gfCNCPoint1[9691] = {X 156.3350, Y 7.0477, Z -1.3333, A 0.000, B 0.000, C 0.000 }
gfCNCPoint1[9692] = {X 157.0515, Y 6.6557, Z -1.3333, A 0.000, B 0.000, C 0.000 }
gfCNCPoint1[9693] = {X 157.8307, Y 6.4112, Z -1.3333, A 0.000, B 0.000, C 0.000 }
gfCNCPoint1[9694] = {X 158.6427, Y 6.3237, Z -1.3333, A 0.000, B 0.000, C 0.000 }
gfCNCPoint1[9695] = {X 159.3760, Y 6.3239, Z -1.3333, A 0.000, B 0.000, C 0.000 }
gfCNCPoint1[9696] = {X 160.2928, Y 6.4383, Z -1.3333, A 0.000, B 0.000, C 0.000 }
gfCNCPoint1[9697] = {X 161.1617, Y 6.7524, Z -1.3333, A 0.000, B 0.000, C 0.000 }
gfCNCPoint1[9698] = {X 161.9398, Y 7.2504, Z -1.3333, A 0.000, B 0.000, C 0.000 }
gfCNCPoint1[9699] = {X 162.5889, Y 7.9079, Z -1.3333, A 0.000, B 0.000, C 0.000 }
gfCNCPoint1[9700] = {X 163.0768, Y 8.6925, Z -1.3333, A 0.000, B 0.000, C 0.000 }
gfCNCPoint1[9701] = {X 163.3795, Y 9.5653, Z -1.3333, A 0.000, B 0.000, C 0.000 }
gfCNCPoint1[9702] = {X 163.4821, Y 10.4835, Z -1.3333, A 0.000, B 0.000, C 0.000 }
gfCNCPoint1[9703] = {X 163.4821, Y 17.4615, Z -1.3333, A 0.000, B 0.000, C 0.000 }
gfCNCPoint1[9704] = {X 163.3795, Y 18.3798, Z -1.3333, A 0.000, B 0.000, C 0.000 }
gfCNCPoint1[9705] = {X 163.0767, Y 19.2527, Z -1.3333, A 0.000, B 0.000, C 0.000 }
gfCNCPoint1[9706] = {X 162.5887, Y 20.0373, Z -1.3333, A 0.000, B 0.000, C 0.000 }
gfCNCPoint1[9707] = {X 161.9396, Y 20.6948, Z -1.3333, A 0.000, B 0.000, C 0.000 }
gfCNCPoint1[9708] = {X 161.1613, Y 21.1929, Z -1.3333, A 0.000, B 0.000, C 0.000 }
gfCNCPoint1[9709] = {X 160.2923, Y 21.5068, Z -1.3333, A 0.000, B 0.000, C 0.000 }
gfCNCPoint1[9710] = {X 159.3755, Y 21.6212, Z -1.3333, A 0.000, B 0.000, C 0.000 }
gfCNCPoint1[9711] = {X 158.6798, Y 21.6215, Z -1.3333, A 0.000, B 0.000, C 0.000 }
gfCNCPoint1[9712] = {X 157.8558, Y 21.5356, Z -1.3333, A 0.000, B 0.000, C 0.000 }
gfCNCPoint1[9713] = {X 157.0647, Y 21.2896, Z -1.3333, A 0.000, B 0.000, C 0.000 }
gfCNCPoint1[9714] = {X 156.3373, Y 20.8931, Z -1.3333, A 0.000, B 0.000, C 0.000 }
gfCNCPoint1[9715] = {X 155.7019, Y 20.3615, Z -1.3333, A 0.000, B 0.000, C 0.000 }
gfCNCPoint1[9716] = {X 155.1831, Y 19.7156, Z -1.3333, A 0.000, B 0.000, C 0.000 }
gfCNCPoint1[9717] = {X 152.1155, Y 19.7172, Z -1.3333, A 0.000, B 0.000, C 0.000 }
gfCNCPoint1[9718] = {X 152.1138, Y 40.9370, Z -1.3333, A 0.000, B 0.000, C 0.000 }
gfCNCPoint1[9719] = {X 152.6210, Y 41.4829, Z -1.3333, A 0.000, B 0.000, C 0.000 }
gfCNCPoint1[9720] = {X 152.7111, Y 41.5906, Z -1.3333, A 0.000, B 0.000, C 0.000 }
gfCNCPoint1[9721] = {X 153.2166, Y 42.3853, Z -1.3333, A 0.000, B 0.000, C 0.000 }
gfCNCPoint1[9722] = {X 153.5326, Y 43.2727, Z -1.3333, A 0.000, B 0.000, C 0.000 }
gfCNCPoint1[9723] = {X 153.6431, Y 44.2081, Z -1.3333, A 0.000, B 0.000, C 0.000 }
gfCNCPoint1[9724] = {X 153.6429, Y 45.0400, Z -1.3333, A 0.000, B 0.000, C 0.000 }
gfCNCPoint1[9725] = {X 153.5310, Y 45.9591, Z -1.3333, A 0.000, B 0.000, C 0.000 }
gfCNCPoint1[9726] = {X 153.2186, Y 46.8306, Z -1.3333, A 0.000, B 0.000, C 0.000 }
gfCNCPoint1[9727] = {X 152.7212, Y 47.6115, Z -1.3333, A 0.000, B 0.000, C 0.000 }
gfCNCPoint1[9728] = {X 152.0634, Y 48.2631, Z -1.3333, A 0.000, B 0.000, C 0.000 }
gfCNCPoint1[9729] = {X 151.2778, Y 48.7530, Z -1.3333, A 0.000, B 0.000, C 0.000 }
gfCNCPoint1[9730] = {X 150.4032, Y 49.0570, Z -1.3333, A 0.000, B 0.000, C 0.000 }
gfCNCPoint1[9731] = {X 149.4831, Y 49.1600, Z -1.3333, A 0.000, B 0.000, C 0.000 }
gfCNCPoint1[9732] = {X 143.0396, Y 49.1600, Z -1.3333, A 0.000, B 0.000, C 0.000 }
gfCNCPoint1[9733] = {X 142.1185, Y 49.0567, Z -1.3333, A 0.000, B 0.000, C 0.000 }
gfCNCPoint1[9734] = {X 141.2432, Y 48.7521, Z -1.3333, A 0.000, B 0.000, C 0.000 }
gfCNCPoint1[9735] = {X 140.4570, Y 48.2612, Z -1.3333, A 0.000, B 0.000, C 0.000 }
gfCNCPoint1[9736] = {X 139.7990, Y 47.6084, Z -1.3333, A 0.000, B 0.000, C 0.000 }
gfCNCPoint1[9737] = {X 139.3019, Y 46.8261, Z -1.3333, A 0.000, B 0.000, C 0.000 }
gfCNCPoint1[9738] = {X 138.9903, Y 45.9532, Z -1.3333, A 0.000, B 0.000, C 0.000 }
gfCNCPoint1[9739] = {X 138.8798, Y 45.0329, Z -1.3333, A 0.000, B 0.000, C 0.000 }
gfCNCPoint1[9740] = {X 138.8800, Y 44.1516, Z -1.3333, A 0.000, B 0.000, C 0.000 }
gfCNCPoint1[9741] = {X 138.9906, Y 43.2545, Z -1.3333, A 0.000, B 0.000, C 0.000 }
gfCNCPoint1[9742] = {X 139.2922, Y 42.4026, Z -1.3333, A 0.000, B 0.000, C 0.000 }
gfCNCPoint1[9743] = {X 139.7708, Y 41.6358, Z -1.3333, A 0.000, B 0.000, C 0.000 }
gfCNCPoint1[9744] = {X 140.4036, Y 40.9906, Z -1.3333, A 0.000, B 0.000, C 0.000 }
gfCNCPoint1[9745] = {X 140.4036, Y 30.3961, Z -1.3333, A 0.000, B 0.000, C 0.000 }
gfCNCPoint1[9746] = {X 136.4036, Y 30.3961, Z -1.3333, A 0.000, B 0.000, C 0.000 }
gfCNCPoint1[9747] = {X 140.4836, Y 30.3961, Z -1.3333, A 0.000, B 0.000, C 0.000 }
gfCNCPoint1[9748] = {X 140.4836, Y 19.6366, Z -1.3333, A 0.000, B 0.000, C 0.000 }
gfCNCPoint1[9749] = {X 137.2908, Y 19.6355, Z -1.3333, A 0.000, B 0.000, C 0.000 }
gfCNCPoint1[9750] = {X 137.2218, Y 19.7475, Z -1.3333, A 0.000, B 0.000, C 0.000 }
gfCNCPoint1[9751] = {X 136.5756, Y 20.4907, Z -1.3333, A 0.000, B 0.000, C 0.000 }
gfCNCPoint1[9752] = {X 135.7702, Y 21.0573, Z -1.3333, A 0.000, B 0.000, C 0.000 }
gfCNCPoint1[9753] = {X 134.8524, Y 21.4145, Z -1.3333, A 0.000, B 0.000, C 0.000 }
gfCNCPoint1[9754] = {X 133.8758, Y 21.5414, Z -1.3333, A 0.000, B 0.000, C 0.000 }
gfCNCPoint1[9755] = {X 133.2006, Y 21.5415, Z -1.3333, A 0.000, B 0.000, C 0.000 }
gfCNCPoint1[9756] = {X 132.2928, Y 21.4392, Z -1.3333, A 0.000, B 0.000, C 0.000 }
gfCNCPoint1[9757] = {X 131.4304, Y 21.1375, Z -1.3333, A 0.000, B 0.000, C 0.000 }
gfCNCPoint1[9758] = {X 130.6568, Y 20.6514, Z -1.3333, A 0.000, B 0.000, C 0.000 }
gfCNCPoint1[9759] = {X 130.0108, Y 20.0054, Z -1.3333, A 0.000, B 0.000, C 0.000 }
gfCNCPoint1[9760] = {X 129.5247, Y 19.2318, Z -1.3333, A 0.000, B 0.000, C 0.000 }
gfCNCPoint1[9761] = {X 129.2229, Y 18.3694, Z -1.3333, A 0.000, B 0.000, C 0.000 }
gfCNCPoint1[9762] = {X 129.1206, Y 17.4615, Z -1.3333, A 0.000, B 0.000, C 0.000 }
gfCNCPoint1[9763] = {X 129.1206, Y 10.4835, Z -1.3333, A 0.000, B 0.000, C 0.000 }
gfCNCPoint1[9764] = {X 129.2215, Y 9.5820, Z -1.3333, A 0.000, B 0.000, C 0.000 }
gfCNCPoint1[9765] = {X 129.5191, Y 8.7250, Z -1.3333, A 0.000, B 0.000, C 0.000 }
gfCNCPoint1[9766] = {X 129.9986, Y 7.9550, Z -1.3333, A 0.000, B 0.000, C 0.000 }
gfCNCPoint1[9767] = {X 130.6365, Y 7.3099, Z -1.3333, A 0.000, B 0.000, C 0.000 }
gfCNCPoint1[9768] = {X 131.4011, Y 6.8218, Z -1.3333, A 0.000, B 0.000, C 0.000 }
gfCNCPoint1[9769] = {X 132.2547, Y 6.5147, Z -1.3333, A 0.000, B 0.000, C 0.000 }
gfCNCPoint1[9770] = {X 133.1551, Y 6.4038, Z -1.3333, A 0.000, B 0.000, C 0.000 }
gfCNCPoint1[9771] = {X 133.8841, Y 6.4037, Z -1.3333, A 0.000, B 0.000, C 0.000 }
gfCNCPoint1[9772] = {X 134.6877, Y 6.4920, Z -1.3333, A 0.000, B 0.000, C 0.000 }
gfCNCPoint1[9773] = {X 135.4580, Y 6.7370, Z -1.3333, A 0.000, B 0.000, C 0.000 }
gfCNCPoint1[9774] = {X 136.1649, Y 7.1291, Z -1.3333, A 0.000, B 0.000, C 0.000 }
gfCNCPoint1[9775] = {X 136.7806, Y 7.6528, Z -1.3333, A 0.000, B 0.000, C 0.000 }
gfCNCPoint1[9776] = {X 137.2810, Y 8.2877, Z -1.3333, A 0.000, B 0.000, C 0.000 }
gfCNCPoint1[9777] = {X 155.2410, Y 8.2888, Z -1.3333, A 0.000, B 0.000, C 0.000 }
gfCNCPoint1[9778] = {X 155.2864, Y 8.2192, Z -1.3333, A 0.000, B 0.000, C 0.000 }
gfCNCPoint1[9779] = {X 155.3332, Y 8.1507, Z -1.3333, A 0.000, B 0.000, C 0.000 }
gfCNCPoint1[9780] = {X 155.9783, Y 7.4266, Z -1.3333, A 0.000, B 0.000, C 0.000 }
gfCNCPoint1[9781] = {X 156.7761, Y 6.8752, Z -1.3333, A 0.000, B 0.000, C 0.000 }
gfCNCPoint1[9782] = {X 157.6815, Y 6.5277, Z -1.3333, A 0.000, B 0.000, C 0.000 }
gfCNCPoint1[9783] = {X 158.6434, Y 6.4037, Z -1.3333, A 0.000, B 0.000, C 0.000 }
gfCNCPoint1[9784] = {X 159.3750, Y 6.4039, Z -1.3333, A 0.000, B 0.000, C 0.000 }
gfCNCPoint1[9785] = {X 160.2741, Y 6.5161, Z -1.3333, A 0.000, B 0.000, C 0.000 }
gfCNCPoint1[9786] = {X 161.1263, Y 6.8241, Z -1.3333, A 0.000, B 0.000, C 0.000 }
gfCNCPoint1[9787] = {X 161.8895, Y 7.3126, Z -1.3333, A 0.000, B 0.000, C 0.000 }
gfCNCPoint1[9788] = {X 162.5260, Y 7.9574, Z -1.3333, A 0.000, B 0.000, C 0.000 }
gfCNCPoint1[9789] = {X 163.0046, Y 8.7269, Z -1.3333, A 0.000, B 0.000, C 0.000 }
gfCNCPoint1[9790] = {X 163.3015, Y 9.5830, Z -1.3333, A 0.000, B 0.000, C 0.000 }
gfCNCPoint1[9791] = {X 163.4021, Y 10.4835, Z -1.3333, A 0.000, B 0.000, C 0.000 }
gfCNCPoint1[9792] = {X 163.4021, Y 17.4615, Z -1.3333, A 0.000, B 0.000, C 0.000 }
gfCNCPoint1[9793] = {X 163.3015, Y 18.3621, Z -1.3333, A 0.000, B 0.000, C 0.000 }
gfCNCPoint1[9794] = {X 163.0046, Y 19.2182, Z -1.3333, A 0.000, B 0.000, C 0.000 }
gfCNCPoint1[9795] = {X 162.5260, Y 19.9876, Z -1.3333, A 0.000, B 0.000, C 0.000 }
gfCNCPoint1[9796] = {X 161.8895, Y 20.6325, Z -1.3333, A 0.000, B 0.000, C 0.000 }
gfCNCPoint1[9797] = {X 161.1263, Y 21.1209, Z -1.3333, A 0.000, B 0.000, C 0.000 }
gfCNCPoint1[9798] = {X 160.2741, Y 21.4289, Z -1.3333, A 0.000, B 0.000, C 0.000 }
gfCNCPoint1[9799] = {X 159.3750, Y 21.5412, Z -1.3333, A 0.000, B 0.000, C 0.000 }
gfCNCPoint1[9800] = {X 158.6802, Y 21.5415, Z -1.3333, A 0.000, B 0.000, C 0.000 }
gfCNCPoint1[9801] = {X 157.8634, Y 21.4555, Z -1.3333, A 0.000, B 0.000, C 0.000 }
gfCNCPoint1[9802] = {X 157.0800, Y 21.2091, Z -1.3333, A 0.000, B 0.000, C 0.000 }
gfCNCPoint1[9803] = {X 156.3609, Y 20.8123, Z -1.3333, A 0.000, B 0.000, C 0.000 }
gfCNCPoint1[9804] = {X 155.7349, Y 20.2807, Z -1.3333, A 0.000, B 0.000, C 0.000 }
gfCNCPoint1[9805] = {X 155.2267, Y 19.6356, Z -1.3333, A 0.000, B 0.000, C 0.000 }
gfCNCPoint1[9806] = {X 152.0355, Y 19.6373, Z -1.3333, A 0.000, B 0.000, C 0.000 }
gfCNCPoint1[9807] = {X 152.0338, Y 40.9684, Z -1.3333, A 0.000, B 0.000, C 0.000 }
gfCNCPoint1[9808] = {X 152.5609, Y 41.5359, Z -1.3333, A 0.000, B 0.000, C 0.000 }
gfCNCPoint1[9809] = {X 152.6492, Y 41.6414, Z -1.3333, A 0.000, B 0.000, C 0.000 }
gfCNCPoint1[9810] = {X 153.1450, Y 42.4209, Z -1.3333, A 0.000, B 0.000, C 0.000 }
gfCNCPoint1[9811] = {X 153.4548, Y 43.2911, Z -1.3333, A 0.000, B 0.000, C 0.000 }
gfCNCPoint1[9812] = {X 153.5631, Y 44.2085, Z -1.3333, A 0.000, B 0.000, C 0.000 }
gfCNCPoint1[9813] = {X 153.5629, Y 45.0392, Z -1.3333, A 0.000, B 0.000, C 0.000 }
gfCNCPoint1[9814] = {X 153.4532, Y 45.9406, Z -1.3333, A 0.000, B 0.000, C 0.000 }
gfCNCPoint1[9815] = {X 153.1468, Y 46.7954, Z -1.3333, A 0.000, B 0.000, C 0.000 }
gfCNCPoint1[9816] = {X 152.6589, Y 47.5613, Z -1.3333, A 0.000, B 0.000, C 0.000 }
gfCNCPoint1[9817] = {X 152.0138, Y 48.2003, Z -1.3333, A 0.000, B 0.000, C 0.000 }
gfCNCPoint1[9818] = {X 151.2432, Y 48.6808, Z -1.3333, A 0.000, B 0.000, C 0.000 }
gfCNCPoint1[9819] = {X 150.3855, Y 48.9789, Z -1.3333, A 0.000, B 0.000, C 0.000 }
gfCNCPoint1[9820] = {X 149.4831, Y 49.0800, Z -1.3333, A 0.000, B 0.000, C 0.000 }
gfCNCPoint1[9821] = {X 143.0396, Y 49.0800, Z -1.3333, A 0.000, B 0.000, C 0.000 }
gfCNCPoint1[9822] = {X 142.1362, Y 48.9787, Z -1.3333, A 0.000, B 0.000, C 0.000 }
gfCNCPoint1[9823] = {X 141.2777, Y 48.6799, Z -1.3333, A 0.000, B 0.000, C 0.000 }
gfCNCPoint1[9824] = {X 140.5066, Y 48.1985, Z -1.3333, A 0.000, B 0.000, C 0.000 }
gfCNCPoint1[9825] = {X 139.8613, Y 47.5582, Z -1.3333, A 0.000, B 0.000, C 0.000 }
gfCNCPoint1[9826] = {X 139.3737, Y 46.7910, Z -1.3333, A 0.000, B 0.000, C 0.000 }
gfCNCPoint1[9827] = {X 139.0682, Y 45.9349, Z -1.3333, A 0.000, B 0.000, C 0.000 }
gfCNCPoint1[9828] = {X 138.9598, Y 45.0323, Z -1.3333, A 0.000, B 0.000, C 0.000 }
gfCNCPoint1[9829] = {X 138.9600, Y 44.1527, Z -1.3333, A 0.000, B 0.000, C 0.000 }
gfCNCPoint1[9830] = {X 139.0706, Y 43.2637, Z -1.3333, A 0.000, B 0.000, C 0.000 }
gfCNCPoint1[9831] = {X 139.3725, Y 42.4203, Z -1.3333, A 0.000, B 0.000, C 0.000 }
gfCNCPoint1[9832] = {X 139.8512, Y 41.6631, Z -1.3333, A 0.000, B 0.000, C 0.000 }
gfCNCPoint1[9833] = {X 140.4836, Y 41.0287, Z -1.3333, A 0.000, B 0.000, C 0.000 }
gfCNCPoint1[9834] = {X 140.4836, Y 30.3961, Z -1.3333, A 0.000, B 0.000, C 0.000 }
gfCNCPoint1[9835] = {X 136.4836, Y 30.3961, Z -1.3333, A 0.000, B 0.000, C 0.000 }
gfCNCPoint1[9836] = {X 140.5636, Y 30.3961, Z -1.3333, A 0.000, B 0.000, C 0.000 }
gfCNCPoint1[9837] = {X 140.5636, Y 19.9565, Z -1.3333, A 0.000, B 0.000, C 0.000 }
gfCNCPoint1[9838] = {X 140.5652, Y 19.5566, Z -1.3333, A 0.000, B 0.000, C 0.000 }
gfCNCPoint1[9839] = {X 137.2663, Y 19.5555, Z -1.3333, A 0.000, B 0.000, C 0.000 }
gfCNCPoint1[9840] = {X 137.2435, Y 19.5597, Z -1.3333, A 0.000, B 0.000, C 0.000 }
gfCNCPoint1[9841] = {X 137.1376, Y 19.7289, Z -1.3333, A 0.000, B 0.000, C 0.000 }
gfCNCPoint1[9842] = {X 136.4981, Y 20.4526, Z -1.3333, A 0.000, B 0.000, C 0.000 }
gfCNCPoint1[9843] = {X 135.7038, Y 21.0020, Z -1.3333, A 0.000, B 0.000, C 0.000 }
gfCNCPoint1[9844] = {X 134.8009, Y 21.3450, Z -1.3333, A 0.000, B 0.000, C 0.000 }
gfCNCPoint1[9845] = {X 133.8421, Y 21.4615, Z -1.3333, A 0.000, B 0.000, C 0.000 }
gfCNCPoint1[9846] = {X 133.2006, Y 21.4615, Z -1.3333, A 0.000, B 0.000, C 0.000 }
gfCNCPoint1[9847] = {X 132.3106, Y 21.3612, Z -1.3333, A 0.000, B 0.000, C 0.000 }
gfCNCPoint1[9848] = {X 131.4651, Y 21.0654, Z -1.3333, A 0.000, B 0.000, C 0.000 }
gfCNCPoint1[9849] = {X 130.7067, Y 20.5889, Z -1.3333, A 0.000, B 0.000, C 0.000 }
gfCNCPoint1[9850] = {X 130.0733, Y 19.9555, Z -1.3333, A 0.000, B 0.000, C 0.000 }
gfCNCPoint1[9851] = {X 129.5968, Y 19.1971, Z -1.3333, A 0.000, B 0.000, C 0.000 }
gfCNCPoint1[9852] = {X 129.3009, Y 18.3516, Z -1.3333, A 0.000, B 0.000, C 0.000 }
gfCNCPoint1[9853] = {X 129.2006, Y 17.4615, Z -1.3333, A 0.000, B 0.000, C 0.000 }
gfCNCPoint1[9854] = {X 129.2006, Y 10.4835, Z -1.3333, A 0.000, B 0.000, C 0.000 }
gfCNCPoint1[9855] = {X 129.3009, Y 9.5934, Z -1.3333, A 0.000, B 0.000, C 0.000 }
gfCNCPoint1[9856] = {X 129.5968, Y 8.7480, Z -1.3333, A 0.000, B 0.000, C 0.000 }
gfCNCPoint1[9857] = {X 130.0733, Y 7.9895, Z -1.3333, A 0.000, B 0.000, C 0.000 }
gfCNCPoint1[9858] = {X 130.7067, Y 7.3562, Z -1.3333, A 0.000, B 0.000, C 0.000 }
gfCNCPoint1[9859] = {X 131.4651, Y 6.8796, Z -1.3333, A 0.000, B 0.000, C 0.000 }
gfCNCPoint1[9860] = {X 132.3106, Y 6.5838, Z -1.3333, A 0.000, B 0.000, C 0.000 }
gfCNCPoint1[9861] = {X 133.2007, Y 6.4835, Z -1.3333, A 0.000, B 0.000, C 0.000 }
gfCNCPoint1[9862] = {X 133.8833, Y 6.4837, Z -1.3333, A 0.000, B 0.000, C 0.000 }
gfCNCPoint1[9863] = {X 134.6796, Y 6.5721, Z -1.3333, A 0.000, B 0.000, C 0.000 }
gfCNCPoint1[9864] = {X 135.4423, Y 6.8175, Z -1.3333, A 0.000, B 0.000, C 0.000 }
gfCNCPoint1[9865] = {X 136.1408, Y 7.2099, Z -1.3333, A 0.000, B 0.000, C 0.000 }
gfCNCPoint1[9866] = {X 136.7471, Y 7.7336, Z -1.3333, A 0.000, B 0.000, C 0.000 }
gfCNCPoint1[9867] = {X 137.2369, Y 8.3677, Z -1.3333, A 0.000, B 0.000, C 0.000 }
gfCNCPoint1[9868] = {X 155.2276, Y 8.3677, Z -1.3333, A 0.000, B 0.000, C 0.000 }
gfCNCPoint1[9869] = {X 155.2814, Y 8.3748, Z -1.3333, A 0.000, B 0.000, C 0.000 }
gfCNCPoint1[9870] = {X 155.3389, Y 8.2848, Z -1.3333, A 0.000, B 0.000, C 0.000 }
gfCNCPoint1[9871] = {X 155.3988, Y 8.1964, Z -1.3333, A 0.000, B 0.000, C 0.000 }
gfCNCPoint1[9872] = {X 156.0381, Y 7.4805, Z -1.3333, A 0.000, B 0.000, C 0.000 }
gfCNCPoint1[9873] = {X 156.8296, Y 6.9374, Z -1.3333, A 0.000, B 0.000, C 0.000 }
gfCNCPoint1[9874] = {X 157.7277, Y 6.5986, Z -1.3333, A 0.000, B 0.000, C 0.000 }
gfCNCPoint1[9875] = {X 158.6806, Y 6.4835, Z -1.3333, A 0.000, B 0.000, C 0.000 }
gfCNCPoint1[9876] = {X 159.3739, Y 6.4839, Z -1.3333, A 0.000, B 0.000, C 0.000 }
gfCNCPoint1[9877] = {X 160.2554, Y 6.5939, Z -1.3333, A 0.000, B 0.000, C 0.000 }
gfCNCPoint1[9878] = {X 161.0909, Y 6.8959, Z -1.3333, A 0.000, B 0.000, C 0.000 }
gfCNCPoint1[9879] = {X 161.8391, Y 7.3747, Z -1.3333, A 0.000, B 0.000, C 0.000 }
gfCNCPoint1[9880] = {X 162.4632, Y 8.0070, Z -1.3333, A 0.000, B 0.000, C 0.000 }
gfCNCPoint1[9881] = {X 162.9324, Y 8.7613, Z -1.3333, A 0.000, B 0.000, C 0.000 }
gfCNCPoint1[9882] = {X 163.2234, Y 9.6007, Z -1.3333, A 0.000, B 0.000, C 0.000 }
gfCNCPoint1[9883] = {X 163.3221, Y 10.4835, Z -1.3333, A 0.000, B 0.000, C 0.000 }
gfCNCPoint1[9884] = {X 163.3221, Y 17.4615, Z -1.3333, A 0.000, B 0.000, C 0.000 }
gfCNCPoint1[9885] = {X 163.2218, Y 18.3516, Z -1.3333, A 0.000, B 0.000, C 0.000 }
gfCNCPoint1[9886] = {X 162.9260, Y 19.1971, Z -1.3333, A 0.000, B 0.000, C 0.000 }
gfCNCPoint1[9887] = {X 162.4494, Y 19.9555, Z -1.3333, A 0.000, B 0.000, C 0.000 }
gfCNCPoint1[9888] = {X 161.8160, Y 20.5889, Z -1.3333, A 0.000, B 0.000, C 0.000 }
gfCNCPoint1[9889] = {X 161.0576, Y 21.0654, Z -1.3333, A 0.000, B 0.000, C 0.000 }
gfCNCPoint1[9890] = {X 160.2121, Y 21.3613, Z -1.3333, A 0.000, B 0.000, C 0.000 }
gfCNCPoint1[9891] = {X 159.3221, Y 21.4615, Z -1.3333, A 0.000, B 0.000, C 0.000 }
gfCNCPoint1[9892] = {X 158.6806, Y 21.4615, Z -1.3333, A 0.000, B 0.000, C 0.000 }
gfCNCPoint1[9893] = {X 157.8711, Y 21.3754, Z -1.3333, A 0.000, B 0.000, C 0.000 }
gfCNCPoint1[9894] = {X 157.0954, Y 21.1287, Z -1.3333, A 0.000, B 0.000, C 0.000 }
gfCNCPoint1[9895] = {X 156.3848, Y 20.7315, Z -1.3333, A 0.000, B 0.000, C 0.000 }
gfCNCPoint1[9896] = {X 155.7683, Y 20.1999, Z -1.3333, A 0.000, B 0.000, C 0.000 }
gfCNCPoint1[9897] = {X 155.2709, Y 19.5555, Z -1.3333, A 0.000, B 0.000, C 0.000 }
gfCNCPoint1[9898] = {X 151.9555, Y 19.5573, Z -1.3333, A 0.000, B 0.000, C 0.000 }
gfCNCPoint1[9899] = {X 151.9538, Y 40.9999, Z -1.3333, A 0.000, B 0.000, C 0.000 }
gfCNCPoint1[9900] = {X 152.5009, Y 41.5888, Z -1.3333, A 0.000, B 0.000, C 0.000 }
gfCNCPoint1[9901] = {X 152.5874, Y 41.6922, Z -1.3333, A 0.000, B 0.000, C 0.000 }
gfCNCPoint1[9902] = {X 153.0733, Y 42.4564, Z -1.3333, A 0.000, B 0.000, C 0.000 }
gfCNCPoint1[9903] = {X 153.3769, Y 43.3096, Z -1.3333, A 0.000, B 0.000, C 0.000 }
gfCNCPoint1[9904] = {X 153.4831, Y 44.2089, Z -1.3333, A 0.000, B 0.000, C 0.000 }
gfCNCPoint1[9905] = {X 153.4829, Y 45.0384, Z -1.3333, A 0.000, B 0.000, C 0.000 }
gfCNCPoint1[9906] = {X 153.3753, Y 45.9222, Z -1.3333, A 0.000, B 0.000, C 0.000 }
gfCNCPoint1[9907] = {X 153.0750, Y 46.7602, Z -1.3333, A 0.000, B 0.000, C 0.000 }
gfCNCPoint1[9908] = {X 152.5967, Y 47.5111, Z -1.3333, A 0.000, B 0.000, C 0.000 }
gfCNCPoint1[9909] = {X 151.9642, Y 48.1376, Z -1.3333, A 0.000, B 0.000, C 0.000 }
gfCNCPoint1[9910] = {X 151.2087, Y 48.6086, Z -1.3333, A 0.000, B 0.000, C 0.000 }
gfCNCPoint1[9911] = {X 150.3678, Y 48.9009, Z -1.3333, A 0.000, B 0.000, C 0.000 }
gfCNCPoint1[9912] = {X 149.4831, Y 49.0000, Z -1.3333, A 0.000, B 0.000, C 0.000 }
gfCNCPoint1[9913] = {X 143.0396, Y 49.0000, Z -1.3333, A 0.000, B 0.000, C 0.000 }
gfCNCPoint1[9914] = {X 142.1495, Y 48.8997, Z -1.3333, A 0.000, B 0.000, C 0.000 }
gfCNCPoint1[9915] = {X 141.3041, Y 48.6039, Z -1.3333, A 0.000, B 0.000, C 0.000 }
gfCNCPoint1[9916] = {X 140.5457, Y 48.1273, Z -1.3333, A 0.000, B 0.000, C 0.000 }
gfCNCPoint1[9917] = {X 139.9123, Y 47.4939, Z -1.3333, A 0.000, B 0.000, C 0.000 }
gfCNCPoint1[9918] = {X 139.4357, Y 46.7355, Z -1.3333, A 0.000, B 0.000, C 0.000 }
gfCNCPoint1[9919] = {X 139.1399, Y 45.8900, Z -1.3333, A 0.000, B 0.000, C 0.000 }
gfCNCPoint1[9920] = {X 139.0396, Y 44.9999, Z -1.3333, A 0.000, B 0.000, C 0.000 }
gfCNCPoint1[9921] = {X 139.0400, Y 44.1538, Z -1.3333, A 0.000, B 0.000, C 0.000 }
gfCNCPoint1[9922] = {X 139.1506, Y 43.2730, Z -1.3333, A 0.000, B 0.000, C 0.000 }
gfCNCPoint1[9923] = {X 139.4528, Y 42.4382, Z -1.3333, A 0.000, B 0.000, C 0.000 }
gfCNCPoint1[9924] = {X 139.9317, Y 41.6907, Z -1.3333, A 0.000, B 0.000, C 0.000 }
gfCNCPoint1[9925] = {X 140.5636, Y 41.0672, Z -1.3333, A 0.000, B 0.000, C 0.000 }
gfCNCPoint1[9926] = {X 140.5636, Y 30.3961, Z -1.3333, A 0.000, B 0.000, C 0.000 }
gfCNCPoint1[9927] = {X 136.4836, Y 30.3961, Z -1.3333, A 0.000, B 0.000, C 0.000 }
gfCNCPoint1[9928] = {X 136.4836, Y 30.3961, Z 1.6667, A 0.000, B 0.000, C 0.000 }
gfCNCPoint1[9929] = {X 136.4836, Y 30.3961, Z 11.0000, A 0.000, B 0.000, C 0.000 }
gfCNCPoint1[9930] = {X 137.6639, Y 74.8937, Z 11.0000, A 0.000, B 0.000, C 0.000 }
gfCNCPoint1[9931] = {X 137.6639, Y 74.8937, Z 1.6667, A 0.000, B 0.000, C 0.000 }
gfCNCPoint1[9932] = {X 137.6639, Y 74.8937, Z -1.3333, A 0.000, B 0.000, C 0.000 }
gfCNCPoint1[9933] = {X 140.6806, Y 77.6408, Z -1.3333, A 0.000, B 0.000, C 0.000 }
gfCNCPoint1[9934] = {X 155.6330, Y 61.2211, Z -1.3333, A 0.000, B 0.000, C 0.000 }
gfCNCPoint1[9935] = {X 155.2777, Y 60.5151, Z -1.3333, A 0.000, B 0.000, C 0.000 }
gfCNCPoint1[9936] = {X 155.0569, Y 59.7562, Z -1.3333, A 0.000, B 0.000, C 0.000 }
gfCNCPoint1[9937] = {X 154.9781, Y 58.9697, Z -1.3333, A 0.000, B 0.000, C 0.000 }
gfCNCPoint1[9938] = {X 154.9780, Y 58.0000, Z -1.3333, A 0.000, B 0.000, C 0.000 }
gfCNCPoint1[9939] = {X 155.0863, Y 57.0387, Z -1.3333, A 0.000, B 0.000, C 0.000 }
gfCNCPoint1[9940] = {X 155.4058, Y 56.1256, Z -1.3333, A 0.000, B 0.000, C 0.000 }
gfCNCPoint1[9941] = {X 155.9204, Y 55.3065, Z -1.3333, A 0.000, B 0.000, C 0.000 }
gfCNCPoint1[9942] = {X 156.6045, Y 54.6225, Z -1.3333, A 0.000, B 0.000, C 0.000 }
gfCNCPoint1[9943] = {X 157.4236, Y 54.1078, Z -1.3333, A 0.000, B 0.000, C 0.000 }
gfCNCPoint1[9944] = {X 158.3367, Y 53.7883, Z -1.3333, A 0.000, B 0.000, C 0.000 }
gfCNCPoint1[9945] = {X 159.2980, Y 53.6800, Z -1.3333, A 0.000, B 0.000, C 0.000 }
gfCNCPoint1[9946] = {X 178.5335, Y 53.6800, Z -1.3333, A 0.000, B 0.000, C 0.000 }
gfCNCPoint1[9947] = {X 179.4948, Y 53.7883, Z -1.3333, A 0.000, B 0.000, C 0.000 }
gfCNCPoint1[9948] = {X 180.4079, Y 54.1078, Z -1.3333, A 0.000, B 0.000, C 0.000 }
gfCNCPoint1[9949] = {X 181.2270, Y 54.6225, Z -1.3333, A 0.000, B 0.000, C 0.000 }
gfCNCPoint1[9950] = {X 181.9110, Y 55.3065, Z -1.3333, A 0.000, B 0.000, C 0.000 }
gfCNCPoint1[9951] = {X 182.4257, Y 56.1256, Z -1.3333, A 0.000, B 0.000, C 0.000 }
gfCNCPoint1[9952] = {X 182.7452, Y 57.0387, Z -1.3333, A 0.000, B 0.000, C 0.000 }
gfCNCPoint1[9953] = {X 182.8535, Y 58.0000, Z -1.3333, A 0.000, B 0.000, C 0.000 }
gfCNCPoint1[9954] = {X 182.8535, Y 58.9342, Z -1.3333, A 0.000, B 0.000, C 0.000 }
gfCNCPoint1[9955] = {X 182.7807, Y 59.7236, Z -1.3333, A 0.000, B 0.000, C 0.000 }
gfCNCPoint1[9956] = {X 182.5649, Y 60.4865, Z -1.3333, A 0.000, B 0.000, C 0.000 }
gfCNCPoint1[9957] = {X 182.2134, Y 61.1970, Z -1.3333, A 0.000, B 0.000, C 0.000 }
gfCNCPoint1[9958] = {X 209.4771, Y 90.9538, Z -1.3333, A 0.000, B 0.000, C 0.000 }
gfCNCPoint1[9959] = {X 210.1356, Y 91.6218, Z -1.3333, A 0.000, B 0.000, C 0.000 }
gfCNCPoint1[9960] = {X 210.8409, Y 92.2402, Z -1.3333, A 0.000, B 0.000, C 0.000 }
gfCNCPoint1[9961] = {X 211.1176, Y 92.4147, Z -1.3333, A 0.000, B 0.000, C 0.000 }
gfCNCPoint1[9962] = {X 211.4280, Y 92.5180, Z -1.3333, A 0.000, B 0.000, C 0.000 }
gfCNCPoint1[9963] = {X 212.4217, Y 92.7023, Z -1.3333, A 0.000, B 0.000, C 0.000 }
gfCNCPoint1[9964] = {X 213.4259, Y 92.8161, Z -1.3333, A 0.000, B 0.000, C 0.000 }
gfCNCPoint1[9965] = {X 214.4655, Y 92.7370, Z -1.3333, A 0.000, B 0.000, C 0.000 }
gfCNCPoint1[9966] = {X 215.5064, Y 92.6769, Z -1.3333, A 0.000, B 0.000, C 0.000 }
gfCNCPoint1[9967] = {X 216.1767, Y 92.6037, Z -1.3333, A 0.000, B 0.000, C 0.000 }
gfCNCPoint1[9968] = {X 216.8222, Y 92.4086, Z -1.3333, A 0.000, B 0.000, C 0.000 }
gfCNCPoint1[9969] = {X 217.4210, Y 92.0984, Z -1.3333, A 0.000, B 0.000, C 0.000 }
gfCNCPoint1[9970] = {X 222.9613, Y 88.5229, Z -1.3333, A 0.000, B 0.000, C 0.000 }
gfCNCPoint1[9971] = {X 245.8295, Y 73.8994, Z -1.3333, A 0.000, B 0.000, C 0.000 }
gfCNCPoint1[9972] = {X 221.6305, Y 64.4024, Z -1.3333, A 0.000, B 0.000, C 0.000 }
gfCNCPoint1[9973] = {X 219.8632, Y 63.8108, Z -1.3333, A 0.000, B 0.000, C 0.000 }
gfCNCPoint1[9974] = {X 218.0398, Y 63.4255, Z -1.3333, A 0.000, B 0.000, C 0.000 }
gfCNCPoint1[9975] = {X 216.1843, Y 63.2516, Z -1.3333, A 0.000, B 0.000, C 0.000 }
gfCNCPoint1[9976] = {X 215.2524, Y 63.1173, Z -1.3333, A 0.000, B 0.000, C 0.000 }
gfCNCPoint1[9977] = {X 214.3717, Y 62.7843, Z -1.3333, A 0.000, B 0.000, C 0.000 }
gfCNCPoint1[9978] = {X 213.5841, Y 62.2685, Z -1.3333, A 0.000, B 0.000, C 0.000 }
gfCNCPoint1[9979] = {X 212.9270, Y 61.5942, Z -1.3333, A 0.000, B 0.000, C 0.000 }
gfCNCPoint1[9980] = {X 212.4315, Y 60.7937, Z -1.3333, A 0.000, B 0.000, C 0.000 }
gfCNCPoint1[9981] = {X 212.1213, Y 59.9048, Z -1.3333, A 0.000, B 0.000, C 0.000 }
gfCNCPoint1[9982] = {X 212.0110, Y 58.9697, Z -1.3333, A 0.000, B 0.000, C 0.000 }
gfCNCPoint1[9983] = {X 212.0108, Y 58.0000, Z -1.3333, A 0.000, B 0.000, C 0.000 }
gfCNCPoint1[9984] = {X 212.1191, Y 57.0387, Z -1.3333, A 0.000, B 0.000, C 0.000 }
gfCNCPoint1[9985] = {X 212.4386, Y 56.1256, Z -1.3333, A 0.000, B 0.000, C 0.000 }
gfCNCPoint1[9986] = {X 212.9533, Y 55.3065, Z -1.3333, A 0.000, B 0.000, C 0.000 }
gfCNCPoint1[9987] = {X 213.6373, Y 54.6225, Z -1.3333, A 0.000, B 0.000, C 0.000 }
gfCNCPoint1[9988] = {X 214.4564, Y 54.1078, Z -1.3333, A 0.000, B 0.000, C 0.000 }
gfCNCPoint1[9989] = {X 215.3695, Y 53.7883, Z -1.3333, A 0.000, B 0.000, C 0.000 }
gfCNCPoint1[9990] = {X 216.3308, Y 53.6800, Z -1.3333, A 0.000, B 0.000, C 0.000 }
gfCNCPoint1[9991] = {X 237.2617, Y 53.6800, Z -1.3333, A 0.000, B 0.000, C 0.000 }
gfCNCPoint1[9992] = {X 238.2230, Y 53.7883, Z -1.3333, A 0.000, B 0.000, C 0.000 }
gfCNCPoint1[9993] = {X 239.1361, Y 54.1078, Z -1.3333, A 0.000, B 0.000, C 0.000 }
gfCNCPoint1[9994] = {X 239.9552, Y 54.6225, Z -1.3333, A 0.000, B 0.000, C 0.000 }
gfCNCPoint1[9995] = {X 240.6392, Y 55.3065, Z -1.3333, A 0.000, B 0.000, C 0.000 }
gfCNCPoint1[9996] = {X 241.1539, Y 56.1256, Z -1.3333, A 0.000, B 0.000, C 0.000 }
gfCNCPoint1[9997] = {X 241.4734, Y 57.0387, Z -1.3333, A 0.000, B 0.000, C 0.000 }
gfCNCPoint1[9998] = {X 241.5817, Y 58.0000, Z -1.3333, A 0.000, B 0.000, C 0.000 }
gfCNCPoint1[9999] = {X 241.5817, Y 58.2330, Z -1.3333, A 0.000, B 0.000, C 0.000 }
gfCNCPoint1[10000] = {X 248.1125, Y 60.7793, Z -1.3333, A 0.000, B 0.000, C 0.000 }
gfCNCPoint1[10001] = {X 275.6342, Y 71.7032, Z -1.3333, A 0.000, B 0.000, C 0.000 }
gfCNCPoint1[10002] = {X 275.6346, Y 63.2125, Z -1.3333, A 0.000, B 0.000, C 0.000 }
gfCNCPoint1[10003] = {X 274.7828, Y 63.0035, Z -1.3333, A 0.000, B 0.000, C 0.000 }
gfCNCPoint1[10004] = {X 273.9907, Y 62.6268, Z -1.3333, A 0.000, B 0.000, C 0.000 }
gfCNCPoint1[10005] = {X 273.2911, Y 62.0978, Z -1.3333, A 0.000, B 0.000, C 0.000 }
gfCNCPoint1[10006] = {X 272.7127, Y 61.4385, Z -1.3333, A 0.000, B 0.000, C 0.000 }
gfCNCPoint1[10007] = {X 272.2794, Y 60.6759, Z -1.3333, A 0.000, B 0.000, C 0.000 }
gfCNCPoint1[10008] = {X 272.0091, Y 59.8415, Z -1.3333, A 0.000, B 0.000, C 0.000 }
gfCNCPoint1[10009] = {X 271.9128, Y 58.9697, Z -1.3333, A 0.000, B 0.000, C 0.000 }
gfCNCPoint1[10010] = {X 271.9127, Y 58.0000, Z -1.3333, A 0.000, B 0.000, C 0.000 }
gfCNCPoint1[10011] = {X 272.0210, Y 57.0387, Z -1.3333, A 0.000, B 0.000, C 0.000 }
gfCNCPoint1[10012] = {X 272.3405, Y 56.1256, Z -1.3333, A 0.000, B 0.000, C 0.000 }
gfCNCPoint1[10013] = {X 272.8552, Y 55.3065, Z -1.3333, A 0.000, B 0.000, C 0.000 }
gfCNCPoint1[10014] = {X 273.5392, Y 54.6225, Z -1.3333, A 0.000, B 0.000, C 0.000 }
gfCNCPoint1[10015] = {X 274.3583, Y 54.1078, Z -1.3333, A 0.000, B 0.000, C 0.000 }
gfCNCPoint1[10016] = {X 275.2714, Y 53.7883, Z -1.3333, A 0.000, B 0.000, C 0.000 }
gfCNCPoint1[10017] = {X 276.2327, Y 53.6800, Z -1.3333, A 0.000, B 0.000, C 0.000 }
gfCNCPoint1[10018] = {X 292.7731, Y 53.6800, Z -1.3333, A 0.000, B 0.000, C 0.000 }
gfCNCPoint1[10019] = {X 293.7344, Y 53.7883, Z -1.3333, A 0.000, B 0.000, C 0.000 }
gfCNCPoint1[10020] = {X 294.6475, Y 54.1078, Z -1.3333, A 0.000, B 0.000, C 0.000 }
gfCNCPoint1[10021] = {X 295.4666, Y 54.6225, Z -1.3333, A 0.000, B 0.000, C 0.000 }
gfCNCPoint1[10022] = {X 296.1506, Y 55.3065, Z -1.3333, A 0.000, B 0.000, C 0.000 }
gfCNCPoint1[10023] = {X 296.6653, Y 56.1256, Z -1.3333, A 0.000, B 0.000, C 0.000 }
gfCNCPoint1[10024] = {X 296.9848, Y 57.0387, Z -1.3333, A 0.000, B 0.000, C 0.000 }
gfCNCPoint1[10025] = {X 297.0931, Y 58.0000, Z -1.3333, A 0.000, B 0.000, C 0.000 }
gfCNCPoint1[10026] = {X 297.0931, Y 58.9352, Z -1.3333, A 0.000, B 0.000, C 0.000 }
gfCNCPoint1[10027] = {X 297.0004, Y 59.8116, Z -1.3333, A 0.000, B 0.000, C 0.000 }
gfCNCPoint1[10028] = {X 296.7325, Y 60.6512, Z -1.3333, A 0.000, B 0.000, C 0.000 }
gfCNCPoint1[10029] = {X 296.3004, Y 61.4193, Z -1.3333, A 0.000, B 0.000, C 0.000 }
gfCNCPoint1[10030] = {X 295.7219, Y 62.0842, Z -1.3333, A 0.000, B 0.000, C 0.000 }
gfCNCPoint1[10031] = {X 295.0210, Y 62.6184, Z -1.3333, A 0.000, B 0.000, C 0.000 }
gfCNCPoint1[10032] = {X 294.2266, Y 62.9999, Z -1.3333, A 0.000, B 0.000, C 0.000 }
gfCNCPoint1[10033] = {X 293.3715, Y 63.2129, Z -1.3333, A 0.000, B 0.000, C 0.000 }
gfCNCPoint1[10034] = {X 293.3840, Y 92.7824, Z -1.3333, A 0.000, B 0.000, C 0.000 }
gfCNCPoint1[10035] = {X 294.2364, Y 92.9998, Z -1.3333, A 0.000, B 0.000, C 0.000 }
gfCNCPoint1[10036] = {X 295.0277, Y 93.3841, Z -1.3333, A 0.000, B 0.000, C 0.000 }
gfCNCPoint1[10037] = {X 295.7256, Y 93.9196, Z -1.3333, A 0.000, B 0.000, C 0.000 }
gfCNCPoint1[10038] = {X 296.3015, Y 94.5846, Z -1.3333, A 0.000, B 0.000, C 0.000 }
gfCNCPoint1[10039] = {X 296.7320, Y 95.3517, Z -1.3333, A 0.000, B 0.000, C 0.000 }
gfCNCPoint1[10040] = {X 296.9995, Y 96.1897, Z -1.3333, A 0.000, B 0.000, C 0.000 }
gfCNCPoint1[10041] = {X 297.0931, Y 97.0644, Z -1.3333, A 0.000, B 0.000, C 0.000 }
gfCNCPoint1[10042] = {X 297.0931, Y 98.0000, Z -1.3333, A 0.000, B 0.000, C 0.000 }
gfCNCPoint1[10043] = {X 296.9848, Y 98.9613, Z -1.3333, A 0.000, B 0.000, C 0.000 }
gfCNCPoint1[10044] = {X 296.6653, Y 99.8744, Z -1.3333, A 0.000, B 0.000, C 0.000 }
gfCNCPoint1[10045] = {X 296.1506, Y 100.6935, Z -1.3333, A 0.000, B 0.000, C 0.000 }
gfCNCPoint1[10046] = {X 295.4666, Y 101.3775, Z -1.3333, A 0.000, B 0.000, C 0.000 }
gfCNCPoint1[10047] = {X 294.6475, Y 101.8922, Z -1.3333, A 0.000, B 0.000, C 0.000 }
gfCNCPoint1[10048] = {X 293.7344, Y 102.2117, Z -1.3333, A 0.000, B 0.000, C 0.000 }
gfCNCPoint1[10049] = {X 292.7731, Y 102.3200, Z -1.3333, A 0.000, B 0.000, C 0.000 }
gfCNCPoint1[10050] = {X 276.2327, Y 102.3200, Z -1.3333, A 0.000, B 0.000, C 0.000 }
gfCNCPoint1[10051] = {X 275.2714, Y 102.2117, Z -1.3333, A 0.000, B 0.000, C 0.000 }
gfCNCPoint1[10052] = {X 274.3583, Y 101.8922, Z -1.3333, A 0.000, B 0.000, C 0.000 }
gfCNCPoint1[10053] = {X 273.5392, Y 101.3775, Z -1.3333, A 0.000, B 0.000, C 0.000 }
gfCNCPoint1[10054] = {X 272.8552, Y 100.6935, Z -1.3333, A 0.000, B 0.000, C 0.000 }
gfCNCPoint1[10055] = {X 272.3405, Y 99.8744, Z -1.3333, A 0.000, B 0.000, C 0.000 }
gfCNCPoint1[10056] = {X 272.0210, Y 98.9613, Z -1.3333, A 0.000, B 0.000, C 0.000 }
gfCNCPoint1[10057] = {X 271.9127, Y 98.0000, Z -1.3333, A 0.000, B 0.000, C 0.000 }
gfCNCPoint1[10058] = {X 271.9127, Y 97.0659, Z -1.3333, A 0.000, B 0.000, C 0.000 }
gfCNCPoint1[10059] = {X 272.0026, Y 96.1891, Z -1.3333, A 0.000, B 0.000, C 0.000 }
gfCNCPoint1[10060] = {X 272.2686, Y 95.3488, Z -1.3333, A 0.000, B 0.000, C 0.000 }
gfCNCPoint1[10061] = {X 272.6996, Y 94.5800, Z -1.3333, A 0.000, B 0.000, C 0.000 }
gfCNCPoint1[10062] = {X 273.2777, Y 93.9147, Z -1.3333, A 0.000, B 0.000, C 0.000 }
gfCNCPoint1[10063] = {X 273.9788, Y 93.3805, Z -1.3333, A 0.000, B 0.000, C 0.000 }
gfCNCPoint1[10064] = {X 274.7737, Y 92.9998, Z -1.3333, A 0.000, B 0.000, C 0.000 }
gfCNCPoint1[10065] = {X 275.6294, Y 92.7883, Z -1.3333, A 0.000, B 0.000, C 0.000 }
gfCNCPoint1[10066] = {X 275.6294, Y 85.5950, Z -1.3333, A 0.000, B 0.000, C 0.000 }
gfCNCPoint1[10067] = {X 262.6395, Y 80.5029, Z -1.3333, A 0.000, B 0.000, C 0.000 }
gfCNCPoint1[10068] = {X 262.2756, Y 80.7317, Z -1.3333, A 0.000, B 0.000, C 0.000 }
gfCNCPoint1[10069] = {X 237.7957, Y 96.5879, Z -1.3333, A 0.000, B 0.000, C 0.000 }
gfCNCPoint1[10070] = {X 237.7998, Y 97.0645, Z -1.3333, A 0.000, B 0.000, C 0.000 }
gfCNCPoint1[10071] = {X 237.7998, Y 98.0000, Z -1.3333, A 0.000, B 0.000, C 0.000 }
gfCNCPoint1[10072] = {X 237.6915, Y 98.9613, Z -1.3333, A 0.000, B 0.000, C 0.000 }
gfCNCPoint1[10073] = {X 237.3720, Y 99.8744, Z -1.3333, A 0.000, B 0.000, C 0.000 }
gfCNCPoint1[10074] = {X 236.8573, Y 100.6935, Z -1.3333, A 0.000, B 0.000, C 0.000 }
gfCNCPoint1[10075] = {X 236.1733, Y 101.3775, Z -1.3333, A 0.000, B 0.000, C 0.000 }
gfCNCPoint1[10076] = {X 235.3542, Y 101.8922, Z -1.3333, A 0.000, B 0.000, C 0.000 }
gfCNCPoint1[10077] = {X 234.4411, Y 102.2117, Z -1.3333, A 0.000, B 0.000, C 0.000 }
gfCNCPoint1[10078] = {X 233.4798, Y 102.3200, Z -1.3333, A 0.000, B 0.000, C 0.000 }
gfCNCPoint1[10079] = {X 214.1790, Y 102.3200, Z -1.3333, A 0.000, B 0.000, C 0.000 }
gfCNCPoint1[10080] = {X 213.7862, Y 102.3021, Z -1.3333, A 0.000, B 0.000, C 0.000 }
gfCNCPoint1[10081] = {X 213.3966, Y 102.2485, Z -1.3333, A 0.000, B 0.000, C 0.000 }
gfCNCPoint1[10082] = {X 213.0070, Y 102.3021, Z -1.3333, A 0.000, B 0.000, C 0.000 }
gfCNCPoint1[10083] = {X 212.6141, Y 102.3200, Z -1.3333, A 0.000, B 0.000, C 0.000 }
gfCNCPoint1[10084] = {X 194.9870, Y 102.3200, Z -1.3333, A 0.000, B 0.000, C 0.000 }
gfCNCPoint1[10085] = {X 194.0257, Y 102.2117, Z -1.3333, A 0.000, B 0.000, C 0.000 }
gfCNCPoint1[10086] = {X 193.1126, Y 101.8922, Z -1.3333, A 0.000, B 0.000, C 0.000 }
gfCNCPoint1[10087] = {X 192.2935, Y 101.3775, Z -1.3333, A 0.000, B 0.000, C 0.000 }
gfCNCPoint1[10088] = {X 191.6094, Y 100.6935, Z -1.3333, A 0.000, B 0.000, C 0.000 }
gfCNCPoint1[10089] = {X 191.0948, Y 99.8744, Z -1.3333, A 0.000, B 0.000, C 0.000 }
gfCNCPoint1[10090] = {X 190.7753, Y 98.9613, Z -1.3333, A 0.000, B 0.000, C 0.000 }
gfCNCPoint1[10091] = {X 190.6670, Y 98.0000, Z -1.3333, A 0.000, B 0.000, C 0.000 }
gfCNCPoint1[10092] = {X 190.6670, Y 97.0659, Z -1.3333, A 0.000, B 0.000, C 0.000 }
gfCNCPoint1[10093] = {X 190.7727, Y 96.1162, Z -1.3333, A 0.000, B 0.000, C 0.000 }
gfCNCPoint1[10094] = {X 191.0846, Y 95.2129, Z -1.3333, A 0.000, B 0.000, C 0.000 }
gfCNCPoint1[10095] = {X 191.5874, Y 94.4003, Z -1.3333, A 0.000, B 0.000, C 0.000 }
gfCNCPoint1[10096] = {X 188.5647, Y 91.1002, Z -1.3333, A 0.000, B 0.000, C 0.000 }
gfCNCPoint1[10097] = {X 150.0898, Y 91.1002, Z -1.3333, A 0.000, B 0.000, C 0.000 }
gfCNCPoint1[10098] = {X 147.1443, Y 94.3635, Z -1.3333, A 0.000, B 0.000, C 0.000 }
gfCNCPoint1[10099] = {X 147.6629, Y 95.1846, Z -1.3333, A 0.000, B 0.000, C 0.000 }
gfCNCPoint1[10100] = {X 147.9866, Y 96.1002, Z -1.3333, A 0.000, B 0.000, C 0.000 }
gfCNCPoint1[10101] = {X 148.0991, Y 97.0648, Z -1.3333, A 0.000, B 0.000, C 0.000 }
gfCNCPoint1[10102] = {X 148.0991, Y 98.0000, Z -1.3333, A 0.000, B 0.000, C 0.000 }
gfCNCPoint1[10103] = {X 147.9908, Y 98.9613, Z -1.3333, A 0.000, B 0.000, C 0.000 }
gfCNCPoint1[10104] = {X 147.6713, Y 99.8744, Z -1.3333, A 0.000, B 0.000, C 0.000 }
gfCNCPoint1[10105] = {X 147.1566, Y 100.6935, Z -1.3333, A 0.000, B 0.000, C 0.000 }
gfCNCPoint1[10106] = {X 146.4726, Y 101.3775, Z -1.3333, A 0.000, B 0.000, C 0.000 }
gfCNCPoint1[10107] = {X 145.6535, Y 101.8922, Z -1.3333, A 0.000, B 0.000, C 0.000 }
gfCNCPoint1[10108] = {X 144.7404, Y 102.2117, Z -1.3333, A 0.000, B 0.000, C 0.000 }
gfCNCPoint1[10109] = {X 143.7791, Y 102.3200, Z -1.3333, A 0.000, B 0.000, C 0.000 }
gfCNCPoint1[10110] = {X 125.0000, Y 102.3200, Z -1.3333, A 0.000, B 0.000, C 0.000 }
gfCNCPoint1[10111] = {X 124.0387, Y 102.2117, Z -1.3333, A 0.000, B 0.000, C 0.000 }
gfCNCPoint1[10112] = {X 123.1256, Y 101.8922, Z -1.3333, A 0.000, B 0.000, C 0.000 }
gfCNCPoint1[10113] = {X 122.3065, Y 101.3775, Z -1.3333, A 0.000, B 0.000, C 0.000 }
gfCNCPoint1[10114] = {X 121.6225, Y 100.6935, Z -1.3333, A 0.000, B 0.000, C 0.000 }
gfCNCPoint1[10115] = {X 121.1078, Y 99.8744, Z -1.3333, A 0.000, B 0.000, C 0.000 }
gfCNCPoint1[10116] = {X 120.7883, Y 98.9613, Z -1.3333, A 0.000, B 0.000, C 0.000 }
gfCNCPoint1[10117] = {X 120.6800, Y 98.0000, Z -1.3333, A 0.000, B 0.000, C 0.000 }
gfCNCPoint1[10118] = {X 120.6800, Y 97.0659, Z -1.3333, A 0.000, B 0.000, C 0.000 }
gfCNCPoint1[10119] = {X 120.7833, Y 96.1269, Z -1.3333, A 0.000, B 0.000, C 0.000 }
gfCNCPoint1[10120] = {X 121.0883, Y 95.2327, Z -1.3333, A 0.000, B 0.000, C 0.000 }
gfCNCPoint1[10121] = {X 121.5803, Y 94.4263, Z -1.3333, A 0.000, B 0.000, C 0.000 }
gfCNCPoint1[10122] = {X 122.2358, Y 93.7460, Z -1.3333, A 0.000, B 0.000, C 0.000 }
gfCNCPoint1[10123] = {X 123.0236, Y 93.2245, Z -1.3333, A 0.000, B 0.000, C 0.000 }
gfCNCPoint1[10124] = {X 123.9059, Y 92.8868, Z -1.3333, A 0.000, B 0.000, C 0.000 }
gfCNCPoint1[10125] = {X 124.8405, Y 92.7489, Z -1.3333, A 0.000, B 0.000, C 0.000 }
gfCNCPoint1[10126] = {X 124.8833, Y 92.7327, Z -1.3333, A 0.000, B 0.000, C 0.000 }
gfCNCPoint1[10127] = {X 124.9280, Y 92.7228, Z -1.3333, A 0.000, B 0.000, C 0.000 }
gfCNCPoint1[10128] = {X 125.4501, Y 92.6453, Z -1.3333, A 0.000, B 0.000, C 0.000 }
gfCNCPoint1[10129] = {X 126.2811, Y 92.5046, Z -1.3333, A 0.000, B 0.000, C 0.000 }
gfCNCPoint1[10130] = {X 127.1010, Y 92.3088, Z -1.3333, A 0.000, B 0.000, C 0.000 }
gfCNCPoint1[10131] = {X 128.3227, Y 91.1567, Z -1.3333, A 0.000, B 0.000, C 0.000 }
gfCNCPoint1[10132] = {X 129.4803, Y 89.9402, Z -1.3333, A 0.000, B 0.000, C 0.000 }
gfCNCPoint1[10133] = {X 140.6806, Y 77.6408, Z -1.3333, A 0.000, B 0.000, C 0.000 }
gfCNCPoint1[10134] = {X 137.7231, Y 74.9476, Z -1.3333, A 0.000, B 0.000, C 0.000 }
gfCNCPoint1[10135] = {X 140.7397, Y 77.6947, Z -1.3333, A 0.000, B 0.000, C 0.000 }
gfCNCPoint1[10136] = {X 155.7332, Y 61.2298, Z -1.3333, A 0.000, B 0.000, C 0.000 }
gfCNCPoint1[10137] = {X 155.3670, Y 60.5232, Z -1.3333, A 0.000, B 0.000, C 0.000 }
gfCNCPoint1[10138] = {X 155.1393, Y 59.7607, Z -1.3333, A 0.000, B 0.000, C 0.000 }
gfCNCPoint1[10139] = {X 155.0581, Y 58.9691, Z -1.3333, A 0.000, B 0.000, C 0.000 }
gfCNCPoint1[10140] = {X 155.0580, Y 58.0000, Z -1.3333, A 0.000, B 0.000, C 0.000 }
gfCNCPoint1[10141] = {X 155.1643, Y 57.0565, Z -1.3333, A 0.000, B 0.000, C 0.000 }
gfCNCPoint1[10142] = {X 155.4778, Y 56.1603, Z -1.3333, A 0.000, B 0.000, C 0.000 }
gfCNCPoint1[10143] = {X 155.9830, Y 55.3564, Z -1.3333, A 0.000, B 0.000, C 0.000 }
gfCNCPoint1[10144] = {X 156.6544, Y 54.6850, Z -1.3333, A 0.000, B 0.000, C 0.000 }
gfCNCPoint1[10145] = {X 157.4583, Y 54.1799, Z -1.3333, A 0.000, B 0.000, C 0.000 }
gfCNCPoint1[10146] = {X 158.3545, Y 53.8663, Z -1.3333, A 0.000, B 0.000, C 0.000 }
gfCNCPoint1[10147] = {X 159.2980, Y 53.7600, Z -1.3333, A 0.000, B 0.000, C 0.000 }
gfCNCPoint1[10148] = {X 178.5335, Y 53.7600, Z -1.3333, A 0.000, B 0.000, C 0.000 }
gfCNCPoint1[10149] = {X 179.4770, Y 53.8663, Z -1.3333, A 0.000, B 0.000, C 0.000 }
gfCNCPoint1[10150] = {X 180.3732, Y 54.1799, Z -1.3333, A 0.000, B 0.000, C 0.000 }
gfCNCPoint1[10151] = {X 181.1771, Y 54.6850, Z -1.3333, A 0.000, B 0.000, C 0.000 }
gfCNCPoint1[10152] = {X 181.8485, Y 55.3564, Z -1.3333, A 0.000, B 0.000, C 0.000 }
gfCNCPoint1[10153] = {X 182.3536, Y 56.1603, Z -1.3333, A 0.000, B 0.000, C 0.000 }
gfCNCPoint1[10154] = {X 182.6672, Y 57.0565, Z -1.3333, A 0.000, B 0.000, C 0.000 }
gfCNCPoint1[10155] = {X 182.7735, Y 58.0000, Z -1.3333, A 0.000, B 0.000, C 0.000 }
gfCNCPoint1[10156] = {X 182.7735, Y 58.9342, Z -1.3333, A 0.000, B 0.000, C 0.000 }
gfCNCPoint1[10157] = {X 182.6984, Y 59.7288, Z -1.3333, A 0.000, B 0.000, C 0.000 }
gfCNCPoint1[10158] = {X 182.4757, Y 60.4951, Z -1.3333, A 0.000, B 0.000, C 0.000 }
gfCNCPoint1[10159] = {X 182.1133, Y 61.2062, Z -1.3333, A 0.000, B 0.000, C 0.000 }
gfCNCPoint1[10160] = {X 209.4181, Y 91.0078, Z -1.3333, A 0.000, B 0.000, C 0.000 }
gfCNCPoint1[10161] = {X 210.0807, Y 91.6800, Z -1.3333, A 0.000, B 0.000, C 0.000 }
gfCNCPoint1[10162] = {X 210.7904, Y 92.3022, Z -1.3333, A 0.000, B 0.000, C 0.000 }
gfCNCPoint1[10163] = {X 211.0834, Y 92.4870, Z -1.3333, A 0.000, B 0.000, C 0.000 }
gfCNCPoint1[10164] = {X 211.4121, Y 92.5964, Z -1.3333, A 0.000, B 0.000, C 0.000 }
gfCNCPoint1[10165] = {X 212.4139, Y 92.7820, Z -1.3333, A 0.000, B 0.000, C 0.000 }
gfCNCPoint1[10166] = {X 213.4262, Y 92.8964, Z -1.3333, A 0.000, B 0.000, C 0.000 }
gfCNCPoint1[10167] = {X 214.4670, Y 92.8171, Z -1.3333, A 0.000, B 0.000, C 0.000 }
gfCNCPoint1[10168] = {X 215.5090, Y 92.7569, Z -1.3333, A 0.000, B 0.000, C 0.000 }
gfCNCPoint1[10169] = {X 216.1936, Y 92.6819, Z -1.3333, A 0.000, B 0.000, C 0.000 }
gfCNCPoint1[10170] = {X 216.8528, Y 92.4825, Z -1.3333, A 0.000, B 0.000, C 0.000 }
gfCNCPoint1[10171] = {X 217.4643, Y 92.1657, Z -1.3333, A 0.000, B 0.000, C 0.000 }
gfCNCPoint1[10172] = {X 223.0046, Y 88.5902, Z -1.3333, A 0.000, B 0.000, C 0.000 }
gfCNCPoint1[10173] = {X 246.0048, Y 73.8823, Z -1.3333, A 0.000, B 0.000, C 0.000 }
gfCNCPoint1[10174] = {X 221.6602, Y 64.3281, Z -1.3333, A 0.000, B 0.000, C 0.000 }
gfCNCPoint1[10175] = {X 219.8842, Y 63.7336, Z -1.3333, A 0.000, B 0.000, C 0.000 }
gfCNCPoint1[10176] = {X 218.0518, Y 63.3464, Z -1.3333, A 0.000, B 0.000, C 0.000 }
gfCNCPoint1[10177] = {X 216.1872, Y 63.1716, Z -1.3333, A 0.000, B 0.000, C 0.000 }
gfCNCPoint1[10178] = {X 215.2725, Y 63.0399, Z -1.3333, A 0.000, B 0.000, C 0.000 }
gfCNCPoint1[10179] = {X 214.4081, Y 62.7131, Z -1.3333, A 0.000, B 0.000, C 0.000 }
gfCNCPoint1[10180] = {X 213.6351, Y 62.2068, Z -1.3333, A 0.000, B 0.000, C 0.000 }
gfCNCPoint1[10181] = {X 212.9901, Y 61.5450, Z -1.3333, A 0.000, B 0.000, C 0.000 }
gfCNCPoint1[10182] = {X 212.5038, Y 60.7593, Z -1.3333, A 0.000, B 0.000, C 0.000 }
gfCNCPoint1[10183] = {X 212.1992, Y 59.8868, Z -1.3333, A 0.000, B 0.000, C 0.000 }
gfCNCPoint1[10184] = {X 212.0910, Y 58.9691, Z -1.3333, A 0.000, B 0.000, C 0.000 }
gfCNCPoint1[10185] = {X 212.0908, Y 58.0000, Z -1.3333, A 0.000, B 0.000, C 0.000 }
gfCNCPoint1[10186] = {X 212.1971, Y 57.0565, Z -1.3333, A 0.000, B 0.000, C 0.000 }
gfCNCPoint1[10187] = {X 212.5107, Y 56.1603, Z -1.3333, A 0.000, B 0.000, C 0.000 }
gfCNCPoint1[10188] = {X 213.0158, Y 55.3564, Z -1.3333, A 0.000, B 0.000, C 0.000 }
gfCNCPoint1[10189] = {X 213.6872, Y 54.6850, Z -1.3333, A 0.000, B 0.000, C 0.000 }
gfCNCPoint1[10190] = {X 214.4911, Y 54.1799, Z -1.3333, A 0.000, B 0.000, C 0.000 }
gfCNCPoint1[10191] = {X 215.3873, Y 53.8663, Z -1.3333, A 0.000, B 0.000, C 0.000 }
gfCNCPoint1[10192] = {X 216.3308, Y 53.7600, Z -1.3333, A 0.000, B 0.000, C 0.000 }
gfCNCPoint1[10193] = {X 237.2617, Y 53.7600, Z -1.3333, A 0.000, B 0.000, C 0.000 }
gfCNCPoint1[10194] = {X 238.2052, Y 53.8663, Z -1.3333, A 0.000, B 0.000, C 0.000 }
gfCNCPoint1[10195] = {X 239.1014, Y 54.1799, Z -1.3333, A 0.000, B 0.000, C 0.000 }
gfCNCPoint1[10196] = {X 239.9053, Y 54.6850, Z -1.3333, A 0.000, B 0.000, C 0.000 }
gfCNCPoint1[10197] = {X 240.5767, Y 55.3564, Z -1.3333, A 0.000, B 0.000, C 0.000 }
gfCNCPoint1[10198] = {X 241.0818, Y 56.1603, Z -1.3333, A 0.000, B 0.000, C 0.000 }
gfCNCPoint1[10199] = {X 241.3954, Y 57.0565, Z -1.3333, A 0.000, B 0.000, C 0.000 }
gfCNCPoint1[10200] = {X 241.5017, Y 58.0000, Z -1.3333, A 0.000, B 0.000, C 0.000 }
gfCNCPoint1[10201] = {X 241.5017, Y 58.2877, Z -1.3333, A 0.000, B 0.000, C 0.000 }
gfCNCPoint1[10202] = {X 248.0832, Y 60.8537, Z -1.3333, A 0.000, B 0.000, C 0.000 }
gfCNCPoint1[10203] = {X 275.7142, Y 71.8210, Z -1.3333, A 0.000, B 0.000, C 0.000 }
gfCNCPoint1[10204] = {X 275.7146, Y 63.1423, Z -1.3333, A 0.000, B 0.000, C 0.000 }
gfCNCPoint1[10205] = {X 274.8659, Y 62.9477, Z -1.3333, A 0.000, B 0.000, C 0.000 }
gfCNCPoint1[10206] = {X 274.0749, Y 62.5839, Z -1.3333, A 0.000, B 0.000, C 0.000 }
gfCNCPoint1[10207] = {X 273.3748, Y 62.0662, Z -1.3333, A 0.000, B 0.000, C 0.000 }
gfCNCPoint1[10208] = {X 272.7953, Y 61.4163, Z -1.3333, A 0.000, B 0.000, C 0.000 }
gfCNCPoint1[10209] = {X 272.3607, Y 60.6618, Z -1.3333, A 0.000, B 0.000, C 0.000 }
gfCNCPoint1[10210] = {X 272.0894, Y 59.8344, Z -1.3333, A 0.000, B 0.000, C 0.000 }
gfCNCPoint1[10211] = {X 271.9928, Y 58.9691, Z -1.3333, A 0.000, B 0.000, C 0.000 }
gfCNCPoint1[10212] = {X 271.9927, Y 58.0000, Z -1.3333, A 0.000, B 0.000, C 0.000 }
gfCNCPoint1[10213] = {X 272.0990, Y 57.0565, Z -1.3333, A 0.000, B 0.000, C 0.000 }
gfCNCPoint1[10214] = {X 272.4126, Y 56.1603, Z -1.3333, A 0.000, B 0.000, C 0.000 }
gfCNCPoint1[10215] = {X 272.9177, Y 55.3564, Z -1.3333, A 0.000, B 0.000, C 0.000 }
gfCNCPoint1[10216] = {X 273.5891, Y 54.6850, Z -1.3333, A 0.000, B 0.000, C 0.000 }
gfCNCPoint1[10217] = {X 274.3930, Y 54.1799, Z -1.3333, A 0.000, B 0.000, C 0.000 }
gfCNCPoint1[10218] = {X 275.2892, Y 53.8663, Z -1.3333, A 0.000, B 0.000, C 0.000 }
gfCNCPoint1[10219] = {X 276.2327, Y 53.7600, Z -1.3333, A 0.000, B 0.000, C 0.000 }
gfCNCPoint1[10220] = {X 292.7731, Y 53.7600, Z -1.3333, A 0.000, B 0.000, C 0.000 }
gfCNCPoint1[10221] = {X 293.7166, Y 53.8663, Z -1.3333, A 0.000, B 0.000, C 0.000 }
gfCNCPoint1[10222] = {X 294.6128, Y 54.1799, Z -1.3333, A 0.000, B 0.000, C 0.000 }
gfCNCPoint1[10223] = {X 295.4167, Y 54.6850, Z -1.3333, A 0.000, B 0.000, C 0.000 }
gfCNCPoint1[10224] = {X 296.0881, Y 55.3564, Z -1.3333, A 0.000, B 0.000, C 0.000 }
gfCNCPoint1[10225] = {X 296.5932, Y 56.1603, Z -1.3333, A 0.000, B 0.000, C 0.000 }
gfCNCPoint1[10226] = {X 296.9068, Y 57.0565, Z -1.3333, A 0.000, B 0.000, C 0.000 }
gfCNCPoint1[10227] = {X 297.0131, Y 58.0000, Z -1.3333, A 0.000, B 0.000, C 0.000 }
gfCNCPoint1[10228] = {X 297.0131, Y 58.9350, Z -1.3333, A 0.000, B 0.000, C 0.000 }
gfCNCPoint1[10229] = {X 296.9201, Y 59.8045, Z -1.3333, A 0.000, B 0.000, C 0.000 }
gfCNCPoint1[10230] = {X 296.6515, Y 60.6368, Z -1.3333, A 0.000, B 0.000, C 0.000 }
gfCNCPoint1[10231] = {X 296.2184, Y 61.3965, Z -1.3333, A 0.000, B 0.000, C 0.000 }
gfCNCPoint1[10232] = {X 295.6393, Y 62.0518, Z -1.3333, A 0.000, B 0.000, C 0.000 }
gfCNCPoint1[10233] = {X 294.9384, Y 62.5749, Z -1.3333, A 0.000, B 0.000, C 0.000 }
gfCNCPoint1[10234] = {X 294.1455, Y 62.9437, Z -1.3333, A 0.000, B 0.000, C 0.000 }
gfCNCPoint1[10235] = {X 293.2939, Y 63.1427, Z -1.3333, A 0.000, B 0.000, C 0.000 }
gfCNCPoint1[10236] = {X 293.3040, Y 92.8519, Z -1.3333, A 0.000, B 0.000, C 0.000 }
gfCNCPoint1[10237] = {X 294.1534, Y 93.0550, Z -1.3333, A 0.000, B 0.000, C 0.000 }
gfCNCPoint1[10238] = {X 294.9437, Y 93.4266, Z -1.3333, A 0.000, B 0.000, C 0.000 }
gfCNCPoint1[10239] = {X 295.6420, Y 93.9510, Z -1.3333, A 0.000, B 0.000, C 0.000 }
gfCNCPoint1[10240] = {X 296.2190, Y 94.6065, Z -1.3333, A 0.000, B 0.000, C 0.000 }
gfCNCPoint1[10241] = {X 296.6508, Y 95.3656, Z -1.3333, A 0.000, B 0.000, C 0.000 }
gfCNCPoint1[10242] = {X 296.9192, Y 96.1966, Z -1.3333, A 0.000, B 0.000, C 0.000 }
gfCNCPoint1[10243] = {X 297.0131, Y 97.0648, Z -1.3333, A 0.000, B 0.000, C 0.000 }
gfCNCPoint1[10244] = {X 297.0131, Y 98.0000, Z -1.3333, A 0.000, B 0.000, C 0.000 }
gfCNCPoint1[10245] = {X 296.9068, Y 98.9435, Z -1.3333, A 0.000, B 0.000, C 0.000 }
gfCNCPoint1[10246] = {X 296.5932, Y 99.8397, Z -1.3333, A 0.000, B 0.000, C 0.000 }
gfCNCPoint1[10247] = {X 296.0881, Y 100.6436, Z -1.3333, A 0.000, B 0.000, C 0.000 }
gfCNCPoint1[10248] = {X 295.4167, Y 101.3150, Z -1.3333, A 0.000, B 0.000, C 0.000 }
gfCNCPoint1[10249] = {X 294.6128, Y 101.8201, Z -1.3333, A 0.000, B 0.000, C 0.000 }
gfCNCPoint1[10250] = {X 293.7166, Y 102.1337, Z -1.3333, A 0.000, B 0.000, C 0.000 }
gfCNCPoint1[10251] = {X 292.7731, Y 102.2400, Z -1.3333, A 0.000, B 0.000, C 0.000 }
gfCNCPoint1[10252] = {X 276.2327, Y 102.2400, Z -1.3333, A 0.000, B 0.000, C 0.000 }
gfCNCPoint1[10253] = {X 275.2892, Y 102.1337, Z -1.3333, A 0.000, B 0.000, C 0.000 }
gfCNCPoint1[10254] = {X 274.3930, Y 101.8201, Z -1.3333, A 0.000, B 0.000, C 0.000 }
gfCNCPoint1[10255] = {X 273.5891, Y 101.3150, Z -1.3333, A 0.000, B 0.000, C 0.000 }
gfCNCPoint1[10256] = {X 272.9177, Y 100.6436, Z -1.3333, A 0.000, B 0.000, C 0.000 }
gfCNCPoint1[10257] = {X 272.4126, Y 99.8397, Z -1.3333, A 0.000, B 0.000, C 0.000 }
gfCNCPoint1[10258] = {X 272.0990, Y 98.9435, Z -1.3333, A 0.000, B 0.000, C 0.000 }
gfCNCPoint1[10259] = {X 271.9927, Y 98.0000, Z -1.3333, A 0.000, B 0.000, C 0.000 }
gfCNCPoint1[10260] = {X 271.9927, Y 97.0659, Z -1.3333, A 0.000, B 0.000, C 0.000 }
gfCNCPoint1[10261] = {X 272.0830, Y 96.1957, Z -1.3333, A 0.000, B 0.000, C 0.000 }
gfCNCPoint1[10262] = {X 272.3499, Y 95.3624, Z -1.3333, A 0.000, B 0.000, C 0.000 }
gfCNCPoint1[10263] = {X 272.7823, Y 94.6018, Z -1.3333, A 0.000, B 0.000, C 0.000 }
gfCNCPoint1[10264] = {X 273.3615, Y 93.9460, Z -1.3333, A 0.000, B 0.000, C 0.000 }
gfCNCPoint1[10265] = {X 274.0630, Y 93.4231, Z -1.3333, A 0.000, B 0.000, C 0.000 }
gfCNCPoint1[10266] = {X 274.8569, Y 93.0553, Z -1.3333, A 0.000, B 0.000, C 0.000 }
gfCNCPoint1[10267] = {X 275.7094, Y 92.8584, Z -1.3333, A 0.000, B 0.000, C 0.000 }
gfCNCPoint1[10268] = {X 275.7094, Y 85.5404, Z -1.3333, A 0.000, B 0.000, C 0.000 }
gfCNCPoint1[10269] = {X 262.6311, Y 80.4137, Z -1.3333, A 0.000, B 0.000, C 0.000 }
gfCNCPoint1[10270] = {X 262.2325, Y 80.6643, Z -1.3333, A 0.000, B 0.000, C 0.000 }
gfCNCPoint1[10271] = {X 237.7153, Y 96.5446, Z -1.3333, A 0.000, B 0.000, C 0.000 }
gfCNCPoint1[10272] = {X 237.7198, Y 97.0649, Z -1.3333, A 0.000, B 0.000, C 0.000 }
gfCNCPoint1[10273] = {X 237.7198, Y 98.0000, Z -1.3333, A 0.000, B 0.000, C 0.000 }
gfCNCPoint1[10274] = {X 237.6135, Y 98.9435, Z -1.3333, A 0.000, B 0.000, C 0.000 }
gfCNCPoint1[10275] = {X 237.2999, Y 99.8397, Z -1.3333, A 0.000, B 0.000, C 0.000 }
gfCNCPoint1[10276] = {X 236.7948, Y 100.6436, Z -1.3333, A 0.000, B 0.000, C 0.000 }
gfCNCPoint1[10277] = {X 236.1234, Y 101.3150, Z -1.3333, A 0.000, B 0.000, C 0.000 }
gfCNCPoint1[10278] = {X 235.3195, Y 101.8201, Z -1.3333, A 0.000, B 0.000, C 0.000 }
gfCNCPoint1[10279] = {X 234.4233, Y 102.1337, Z -1.3333, A 0.000, B 0.000, C 0.000 }
gfCNCPoint1[10280] = {X 233.4798, Y 102.2400, Z -1.3333, A 0.000, B 0.000, C 0.000 }
gfCNCPoint1[10281] = {X 214.1790, Y 102.2400, Z -1.3333, A 0.000, B 0.000, C 0.000 }
gfCNCPoint1[10282] = {X 213.7861, Y 102.2218, Z -1.3333, A 0.000, B 0.000, C 0.000 }
gfCNCPoint1[10283] = {X 213.3966, Y 102.1672, Z -1.3333, A 0.000, B 0.000, C 0.000 }
gfCNCPoint1[10284] = {X 213.0070, Y 102.2218, Z -1.3333, A 0.000, B 0.000, C 0.000 }
gfCNCPoint1[10285] = {X 212.6141, Y 102.2400, Z -1.3333, A 0.000, B 0.000, C 0.000 }
gfCNCPoint1[10286] = {X 194.9870, Y 102.2400, Z -1.3333, A 0.000, B 0.000, C 0.000 }
gfCNCPoint1[10287] = {X 194.0435, Y 102.1337, Z -1.3333, A 0.000, B 0.000, C 0.000 }
gfCNCPoint1[10288] = {X 193.1473, Y 101.8201, Z -1.3333, A 0.000, B 0.000, C 0.000 }
gfCNCPoint1[10289] = {X 192.3434, Y 101.3150, Z -1.3333, A 0.000, B 0.000, C 0.000 }
gfCNCPoint1[10290] = {X 191.6720, Y 100.6436, Z -1.3333, A 0.000, B 0.000, C 0.000 }
gfCNCPoint1[10291] = {X 191.1669, Y 99.8397, Z -1.3333, A 0.000, B 0.000, C 0.000 }
gfCNCPoint1[10292] = {X 190.8533, Y 98.9435, Z -1.3333, A 0.000, B 0.000, C 0.000 }
gfCNCPoint1[10293] = {X 190.7470, Y 98.0000, Z -1.3333, A 0.000, B 0.000, C 0.000 }
gfCNCPoint1[10294] = {X 190.7470, Y 97.0659, Z -1.3333, A 0.000, B 0.000, C 0.000 }
gfCNCPoint1[10295] = {X 190.8557, Y 96.1118, Z -1.3333, A 0.000, B 0.000, C 0.000 }
gfCNCPoint1[10296] = {X 191.1764, Y 95.2065, Z -1.3333, A 0.000, B 0.000, C 0.000 }
gfCNCPoint1[10297] = {X 191.6926, Y 94.3967, Z -1.3333, A 0.000, B 0.000, C 0.000 }
gfCNCPoint1[10298] = {X 188.5999, Y 91.0202, Z -1.3333, A 0.000, B 0.000, C 0.000 }
gfCNCPoint1[10299] = {X 150.0543, Y 91.0202, Z -1.3333, A 0.000, B 0.000, C 0.000 }
gfCNCPoint1[10300] = {X 147.0390, Y 94.3608, Z -1.3333, A 0.000, B 0.000, C 0.000 }
gfCNCPoint1[10301] = {X 147.5710, Y 95.1788, Z -1.3333, A 0.000, B 0.000, C 0.000 }
gfCNCPoint1[10302] = {X 147.9035, Y 96.0962, Z -1.3333, A 0.000, B 0.000, C 0.000 }
gfCNCPoint1[10303] = {X 148.0191, Y 97.0651, Z -1.3333, A 0.000, B 0.000, C 0.000 }
gfCNCPoint1[10304] = {X 148.0191, Y 98.0000, Z -1.3333, A 0.000, B 0.000, C 0.000 }
gfCNCPoint1[10305] = {X 147.9128, Y 98.9435, Z -1.3333, A 0.000, B 0.000, C 0.000 }
gfCNCPoint1[10306] = {X 147.5992, Y 99.8397, Z -1.3333, A 0.000, B 0.000, C 0.000 }
gfCNCPoint1[10307] = {X 147.0941, Y 100.6436, Z -1.3333, A 0.000, B 0.000, C 0.000 }
gfCNCPoint1[10308] = {X 146.4227, Y 101.3150, Z -1.3333, A 0.000, B 0.000, C 0.000 }
gfCNCPoint1[10309] = {X 145.6188, Y 101.8201, Z -1.3333, A 0.000, B 0.000, C 0.000 }
gfCNCPoint1[10310] = {X 144.7226, Y 102.1337, Z -1.3333, A 0.000, B 0.000, C 0.000 }
gfCNCPoint1[10311] = {X 143.7791, Y 102.2400, Z -1.3333, A 0.000, B 0.000, C 0.000 }
gfCNCPoint1[10312] = {X 125.0000, Y 102.2400, Z -1.3333, A 0.000, B 0.000, C 0.000 }
gfCNCPoint1[10313] = {X 124.0565, Y 102.1337, Z -1.3333, A 0.000, B 0.000, C 0.000 }
gfCNCPoint1[10314] = {X 123.1603, Y 101.8201, Z -1.3333, A 0.000, B 0.000, C 0.000 }
gfCNCPoint1[10315] = {X 122.3564, Y 101.3150, Z -1.3333, A 0.000, B 0.000, C 0.000 }
gfCNCPoint1[10316] = {X 121.6850, Y 100.6436, Z -1.3333, A 0.000, B 0.000, C 0.000 }
gfCNCPoint1[10317] = {X 121.1799, Y 99.8397, Z -1.3333, A 0.000, B 0.000, C 0.000 }
gfCNCPoint1[10318] = {X 120.8663, Y 98.9435, Z -1.3333, A 0.000, B 0.000, C 0.000 }
gfCNCPoint1[10319] = {X 120.7600, Y 98.0000, Z -1.3333, A 0.000, B 0.000, C 0.000 }
gfCNCPoint1[10320] = {X 120.7600, Y 97.0659, Z -1.3333, A 0.000, B 0.000, C 0.000 }
gfCNCPoint1[10321] = {X 120.8619, Y 96.1419, Z -1.3333, A 0.000, B 0.000, C 0.000 }
gfCNCPoint1[10322] = {X 121.1628, Y 95.2622, Z -1.3333, A 0.000, B 0.000, C 0.000 }
gfCNCPoint1[10323] = {X 121.6481, Y 94.4693, Z -1.3333, A 0.000, B 0.000, C 0.000 }
gfCNCPoint1[10324] = {X 122.2946, Y 93.8012, Z -1.3333, A 0.000, B 0.000, C 0.000 }
gfCNCPoint1[10325] = {X 123.0711, Y 93.2901, Z -1.3333, A 0.000, B 0.000, C 0.000 }
gfCNCPoint1[10326] = {X 123.9404, Y 92.9605, Z -1.3333, A 0.000, B 0.000, C 0.000 }
gfCNCPoint1[10327] = {X 124.8606, Y 92.8282, Z -1.3333, A 0.000, B 0.000, C 0.000 }
gfCNCPoint1[10328] = {X 124.8990, Y 92.8116, Z -1.3333, A 0.000, B 0.000, C 0.000 }
gfCNCPoint1[10329] = {X 124.9398, Y 92.8019, Z -1.3333, A 0.000, B 0.000, C 0.000 }
gfCNCPoint1[10330] = {X 125.4608, Y 92.7246, Z -1.3333, A 0.000, B 0.000, C 0.000 }
gfCNCPoint1[10331] = {X 126.3063, Y 92.5811, Z -1.3333, A 0.000, B 0.000, C 0.000 }
gfCNCPoint1[10332] = {X 127.1402, Y 92.3810, Z -1.3333, A 0.000, B 0.000, C 0.000 }
gfCNCPoint1[10333] = {X 128.3725, Y 91.2200, Z -1.3333, A 0.000, B 0.000, C 0.000 }
gfCNCPoint1[10334] = {X 129.5397, Y 89.9938, Z -1.3333, A 0.000, B 0.000, C 0.000 }
gfCNCPoint1[10335] = {X 140.7397, Y 77.6947, Z -1.3333, A 0.000, B 0.000, C 0.000 }
gfCNCPoint1[10336] = {X 137.7822, Y 75.0015, Z -1.3333, A 0.000, B 0.000, C 0.000 }
gfCNCPoint1[10337] = {X 140.7989, Y 77.7485, Z -1.3333, A 0.000, B 0.000, C 0.000 }
gfCNCPoint1[10338] = {X 155.8341, Y 61.2378, Z -1.3333, A 0.000, B 0.000, C 0.000 }
gfCNCPoint1[10339] = {X 155.4567, Y 60.5311, Z -1.3333, A 0.000, B 0.000, C 0.000 }
gfCNCPoint1[10340] = {X 155.2218, Y 59.7652, Z -1.3333, A 0.000, B 0.000, C 0.000 }
gfCNCPoint1[10341] = {X 155.1381, Y 58.9684, Z -1.3333, A 0.000, B 0.000, C 0.000 }
gfCNCPoint1[10342] = {X 155.1380, Y 58.0000, Z -1.3333, A 0.000, B 0.000, C 0.000 }
gfCNCPoint1[10343] = {X 155.2423, Y 57.0743, Z -1.3333, A 0.000, B 0.000, C 0.000 }
gfCNCPoint1[10344] = {X 155.5499, Y 56.1950, Z -1.3333, A 0.000, B 0.000, C 0.000 }
gfCNCPoint1[10345] = {X 156.0455, Y 55.4063, Z -1.3333, A 0.000, B 0.000, C 0.000 }
gfCNCPoint1[10346] = {X 156.7042, Y 54.7476, Z -1.3333, A 0.000, B 0.000, C 0.000 }
gfCNCPoint1[10347] = {X 157.4930, Y 54.2520, Z -1.3333, A 0.000, B 0.000, C 0.000 }
gfCNCPoint1[10348] = {X 158.3723, Y 53.9443, Z -1.3333, A 0.000, B 0.000, C 0.000 }
gfCNCPoint1[10349] = {X 159.2980, Y 53.8400, Z -1.3333, A 0.000, B 0.000, C 0.000 }
gfCNCPoint1[10350] = {X 178.5335, Y 53.8400, Z -1.3333, A 0.000, B 0.000, C 0.000 }
gfCNCPoint1[10351] = {X 179.4592, Y 53.9443, Z -1.3333, A 0.000, B 0.000, C 0.000 }
gfCNCPoint1[10352] = {X 180.3385, Y 54.2520, Z -1.3333, A 0.000, B 0.000, C 0.000 }
gfCNCPoint1[10353] = {X 181.1272, Y 54.7476, Z -1.3333, A 0.000, B 0.000, C 0.000 }
gfCNCPoint1[10354] = {X 181.7859, Y 55.4063, Z -1.3333, A 0.000, B 0.000, C 0.000 }
gfCNCPoint1[10355] = {X 182.2815, Y 56.1950, Z -1.3333, A 0.000, B 0.000, C 0.000 }
gfCNCPoint1[10356] = {X 182.5892, Y 57.0743, Z -1.3333, A 0.000, B 0.000, C 0.000 }
gfCNCPoint1[10357] = {X 182.6935, Y 58.0000, Z -1.3333, A 0.000, B 0.000, C 0.000 }
gfCNCPoint1[10358] = {X 182.6935, Y 58.9342, Z -1.3333, A 0.000, B 0.000, C 0.000 }
gfCNCPoint1[10359] = {X 182.6159, Y 59.7338, Z -1.3333, A 0.000, B 0.000, C 0.000 }
gfCNCPoint1[10360] = {X 182.3861, Y 60.5035, Z -1.3333, A 0.000, B 0.000, C 0.000 }
gfCNCPoint1[10361] = {X 182.0126, Y 61.2147, Z -1.3333, A 0.000, B 0.000, C 0.000 }
gfCNCPoint1[10362] = {X 209.3592, Y 91.0619, Z -1.3333, A 0.000, B 0.000, C 0.000 }
gfCNCPoint1[10363] = {X 210.0258, Y 91.7382, Z -1.3333, A 0.000, B 0.000, C 0.000 }
gfCNCPoint1[10364] = {X 210.7399, Y 92.3642, Z -1.3333, A 0.000, B 0.000, C 0.000 }
gfCNCPoint1[10365] = {X 211.0489, Y 92.5591, Z -1.3333, A 0.000, B 0.000, C 0.000 }
gfCNCPoint1[10366] = {X 211.3954, Y 92.6747, Z -1.3333, A 0.000, B 0.000, C 0.000 }
gfCNCPoint1[10367] = {X 212.4057, Y 92.8617, Z -1.3333, A 0.000, B 0.000, C 0.000 }
gfCNCPoint1[10368] = {X 213.4266, Y 92.9767, Z -1.3333, A 0.000, B 0.000, C 0.000 }
gfCNCPoint1[10369] = {X 214.4685, Y 92.8971, Z -1.3333, A 0.000, B 0.000, C 0.000 }
gfCNCPoint1[10370] = {X 215.5117, Y 92.8369, Z -1.3333, A 0.000, B 0.000, C 0.000 }
gfCNCPoint1[10371] = {X 216.2105, Y 92.7601, Z -1.3333, A 0.000, B 0.000, C 0.000 }
gfCNCPoint1[10372] = {X 216.8835, Y 92.5564, Z -1.3333, A 0.000, B 0.000, C 0.000 }
gfCNCPoint1[10373] = {X 217.5077, Y 92.2329, Z -1.3333, A 0.000, B 0.000, C 0.000 }
gfCNCPoint1[10374] = {X 223.0478, Y 88.6576, Z -1.3333, A 0.000, B 0.000, C 0.000 }
gfCNCPoint1[10375] = {X 246.1801, Y 73.8651, Z -1.3333, A 0.000, B 0.000, C 0.000 }
gfCNCPoint1[10376] = {X 221.6899, Y 64.2538, Z -1.3333, A 0.000, B 0.000, C 0.000 }
gfCNCPoint1[10377] = {X 219.9052, Y 63.6564, Z -1.3333, A 0.000, B 0.000, C 0.000 }
gfCNCPoint1[10378] = {X 218.0638, Y 63.2674, Z -1.3333, A 0.000, B 0.000, C 0.000 }
gfCNCPoint1[10379] = {X 216.1900, Y 63.0917, Z -1.3333, A 0.000, B 0.000, C 0.000 }
gfCNCPoint1[10380] = {X 215.2926, Y 62.9624, Z -1.3333, A 0.000, B 0.000, C 0.000 }
gfCNCPoint1[10381] = {X 214.4445, Y 62.6418, Z -1.3333, A 0.000, B 0.000, C 0.000 }
gfCNCPoint1[10382] = {X 213.6860, Y 62.1451, Z -1.3333, A 0.000, B 0.000, C 0.000 }
gfCNCPoint1[10383] = {X 213.0532, Y 61.4958, Z -1.3333, A 0.000, B 0.000, C 0.000 }
gfCNCPoint1[10384] = {X 212.5760, Y 60.7249, Z -1.3333, A 0.000, B 0.000, C 0.000 }
gfCNCPoint1[10385] = {X 212.2772, Y 59.8688, Z -1.3333, A 0.000, B 0.000, C 0.000 }
gfCNCPoint1[10386] = {X 212.1710, Y 58.9684, Z -1.3333, A 0.000, B 0.000, C 0.000 }
gfCNCPoint1[10387] = {X 212.1708, Y 58.0000, Z -1.3333, A 0.000, B 0.000, C 0.000 }
gfCNCPoint1[10388] = {X 212.2751, Y 57.0743, Z -1.3333, A 0.000, B 0.000, C 0.000 }
gfCNCPoint1[10389] = {X 212.5828, Y 56.1950, Z -1.3333, A 0.000, B 0.000, C 0.000 }
gfCNCPoint1[10390] = {X 213.0784, Y 55.4063, Z -1.3333, A 0.000, B 0.000, C 0.000 }
gfCNCPoint1[10391] = {X 213.7371, Y 54.7476, Z -1.3333, A 0.000, B 0.000, C 0.000 }
gfCNCPoint1[10392] = {X 214.5259, Y 54.2520, Z -1.3333, A 0.000, B 0.000, C 0.000 }
gfCNCPoint1[10393] = {X 215.4051, Y 53.9443, Z -1.3333, A 0.000, B 0.000, C 0.000 }
gfCNCPoint1[10394] = {X 216.3308, Y 53.8400, Z -1.3333, A 0.000, B 0.000, C 0.000 }
gfCNCPoint1[10395] = {X 237.2617, Y 53.8400, Z -1.3333, A 0.000, B 0.000, C 0.000 }
gfCNCPoint1[10396] = {X 238.1874, Y 53.9443, Z -1.3333, A 0.000, B 0.000, C 0.000 }
gfCNCPoint1[10397] = {X 239.0666, Y 54.2520, Z -1.3333, A 0.000, B 0.000, C 0.000 }
gfCNCPoint1[10398] = {X 239.8554, Y 54.7476, Z -1.3333, A 0.000, B 0.000, C 0.000 }
gfCNCPoint1[10399] = {X 240.5141, Y 55.4063, Z -1.3333, A 0.000, B 0.000, C 0.000 }
gfCNCPoint1[10400] = {X 241.0097, Y 56.1950, Z -1.3333, A 0.000, B 0.000, C 0.000 }
gfCNCPoint1[10401] = {X 241.3174, Y 57.0743, Z -1.3333, A 0.000, B 0.000, C 0.000 }
gfCNCPoint1[10402] = {X 241.4217, Y 58.0000, Z -1.3333, A 0.000, B 0.000, C 0.000 }
gfCNCPoint1[10403] = {X 241.4217, Y 58.3424, Z -1.3333, A 0.000, B 0.000, C 0.000 }
gfCNCPoint1[10404] = {X 248.0539, Y 60.9282, Z -1.3333, A 0.000, B 0.000, C 0.000 }
gfCNCPoint1[10405] = {X 275.7942, Y 71.9388, Z -1.3333, A 0.000, B 0.000, C 0.000 }
gfCNCPoint1[10406] = {X 275.7946, Y 63.0709, Z -1.3333, A 0.000, B 0.000, C 0.000 }
gfCNCPoint1[10407] = {X 275.6923, Y 63.0588, Z -1.3333, A 0.000, B 0.000, C 0.000 }
gfCNCPoint1[10408] = {X 275.5903, Y 63.0442, Z -1.3333, A 0.000, B 0.000, C 0.000 }
gfCNCPoint1[10409] = {X 274.6526, Y 62.7823, Z -1.3333, A 0.000, B 0.000, C 0.000 }
gfCNCPoint1[10410] = {X 273.8014, Y 62.3096, Z -1.3333, A 0.000, B 0.000, C 0.000 }
gfCNCPoint1[10411] = {X 273.0834, Y 61.6520, Z -1.3333, A 0.000, B 0.000, C 0.000 }
gfCNCPoint1[10412] = {X 272.5379, Y 60.8456, Z -1.3333, A 0.000, B 0.000, C 0.000 }
gfCNCPoint1[10413] = {X 272.1948, Y 59.9344, Z -1.3333, A 0.000, B 0.000, C 0.000 }
gfCNCPoint1[10414] = {X 272.0728, Y 58.9684, Z -1.3333, A 0.000, B 0.000, C 0.000 }
gfCNCPoint1[10415] = {X 272.0727, Y 58.0000, Z -1.3333, A 0.000, B 0.000, C 0.000 }
gfCNCPoint1[10416] = {X 272.1770, Y 57.0743, Z -1.3333, A 0.000, B 0.000, C 0.000 }
gfCNCPoint1[10417] = {X 272.4847, Y 56.1950, Z -1.3333, A 0.000, B 0.000, C 0.000 }
gfCNCPoint1[10418] = {X 272.9803, Y 55.4063, Z -1.3333, A 0.000, B 0.000, C 0.000 }
gfCNCPoint1[10419] = {X 273.6390, Y 54.7476, Z -1.3333, A 0.000, B 0.000, C 0.000 }
gfCNCPoint1[10420] = {X 274.4277, Y 54.2520, Z -1.3333, A 0.000, B 0.000, C 0.000 }
gfCNCPoint1[10421] = {X 275.3070, Y 53.9443, Z -1.3333, A 0.000, B 0.000, C 0.000 }
gfCNCPoint1[10422] = {X 276.2327, Y 53.8400, Z -1.3333, A 0.000, B 0.000, C 0.000 }
gfCNCPoint1[10423] = {X 292.7731, Y 53.8400, Z -1.3333, A 0.000, B 0.000, C 0.000 }
gfCNCPoint1[10424] = {X 293.6988, Y 53.9443, Z -1.3333, A 0.000, B 0.000, C 0.000 }
gfCNCPoint1[10425] = {X 294.5780, Y 54.2520, Z -1.3333, A 0.000, B 0.000, C 0.000 }
gfCNCPoint1[10426] = {X 295.3668, Y 54.7476, Z -1.3333, A 0.000, B 0.000, C 0.000 }
gfCNCPoint1[10427] = {X 296.0255, Y 55.4063, Z -1.3333, A 0.000, B 0.000, C 0.000 }
gfCNCPoint1[10428] = {X 296.5211, Y 56.1950, Z -1.3333, A 0.000, B 0.000, C 0.000 }
gfCNCPoint1[10429] = {X 296.8288, Y 57.0743, Z -1.3333, A 0.000, B 0.000, C 0.000 }
gfCNCPoint1[10430] = {X 296.9331, Y 58.0000, Z -1.3333, A 0.000, B 0.000, C 0.000 }
gfCNCPoint1[10431] = {X 296.9331, Y 58.9347, Z -1.3333, A 0.000, B 0.000, C 0.000 }
gfCNCPoint1[10432] = {X 296.8149, Y 59.9063, Z -1.3333, A 0.000, B 0.000, C 0.000 }
gfCNCPoint1[10433] = {X 296.4739, Y 60.8237, Z -1.3333, A 0.000, B 0.000, C 0.000 }
gfCNCPoint1[10434] = {X 295.9288, Y 61.6366, Z -1.3333, A 0.000, B 0.000, C 0.000 }
gfCNCPoint1[10435] = {X 295.2095, Y 62.3003, Z -1.3333, A 0.000, B 0.000, C 0.000 }
gfCNCPoint1[10436] = {X 294.3555, Y 62.7784, Z -1.3333, A 0.000, B 0.000, C 0.000 }
gfCNCPoint1[10437] = {X 293.4136, Y 63.0447, Z -1.3333, A 0.000, B 0.000, C 0.000 }
gfCNCPoint1[10438] = {X 293.3174, Y 63.0589, Z -1.3333, A 0.000, B 0.000, C 0.000 }
gfCNCPoint1[10439] = {X 293.2209, Y 63.0709, Z -1.3333, A 0.000, B 0.000, C 0.000 }
gfCNCPoint1[10440] = {X 293.2114, Y 63.1623, Z -1.3333, A 0.000, B 0.000, C 0.000 }
gfCNCPoint1[10441] = {X 293.2241, Y 92.9225, Z -1.3333, A 0.000, B 0.000, C 0.000 }
gfCNCPoint1[10442] = {X 293.3186, Y 92.9346, Z -1.3333, A 0.000, B 0.000, C 0.000 }
gfCNCPoint1[10443] = {X 293.4129, Y 92.9488, Z -1.3333, A 0.000, B 0.000, C 0.000 }
gfCNCPoint1[10444] = {X 294.3544, Y 93.2178, Z -1.3333, A 0.000, B 0.000, C 0.000 }
gfCNCPoint1[10445] = {X 295.2079, Y 93.6977, Z -1.3333, A 0.000, B 0.000, C 0.000 }
gfCNCPoint1[10446] = {X 295.9268, Y 94.3624, Z -1.3333, A 0.000, B 0.000, C 0.000 }
gfCNCPoint1[10447] = {X 296.4719, Y 95.1758, Z -1.3333, A 0.000, B 0.000, C 0.000 }
gfCNCPoint1[10448] = {X 296.8136, Y 96.0934, Z -1.3333, A 0.000, B 0.000, C 0.000 }
gfCNCPoint1[10449] = {X 296.9331, Y 97.0653, Z -1.3333, A 0.000, B 0.000, C 0.000 }
gfCNCPoint1[10450] = {X 296.9331, Y 98.0000, Z -1.3333, A 0.000, B 0.000, C 0.000 }
gfCNCPoint1[10451] = {X 296.8288, Y 98.9257, Z -1.3333, A 0.000, B 0.000, C 0.000 }
gfCNCPoint1[10452] = {X 296.5211, Y 99.8050, Z -1.3333, A 0.000, B 0.000, C 0.000 }
gfCNCPoint1[10453] = {X 296.0255, Y 100.5937, Z -1.3333, A 0.000, B 0.000, C 0.000 }
gfCNCPoint1[10454] = {X 295.3668, Y 101.2524, Z -1.3333, A 0.000, B 0.000, C 0.000 }
gfCNCPoint1[10455] = {X 294.5780, Y 101.7480, Z -1.3333, A 0.000, B 0.000, C 0.000 }
gfCNCPoint1[10456] = {X 293.6988, Y 102.0557, Z -1.3333, A 0.000, B 0.000, C 0.000 }
gfCNCPoint1[10457] = {X 292.7731, Y 102.1600, Z -1.3333, A 0.000, B 0.000, C 0.000 }
gfCNCPoint1[10458] = {X 276.2327, Y 102.1600, Z -1.3333, A 0.000, B 0.000, C 0.000 }
gfCNCPoint1[10459] = {X 275.3070, Y 102.0557, Z -1.3333, A 0.000, B 0.000, C 0.000 }
gfCNCPoint1[10460] = {X 274.4277, Y 101.7480, Z -1.3333, A 0.000, B 0.000, C 0.000 }
gfCNCPoint1[10461] = {X 273.6390, Y 101.2524, Z -1.3333, A 0.000, B 0.000, C 0.000 }
gfCNCPoint1[10462] = {X 272.9803, Y 100.5937, Z -1.3333, A 0.000, B 0.000, C 0.000 }
gfCNCPoint1[10463] = {X 272.4847, Y 99.8050, Z -1.3333, A 0.000, B 0.000, C 0.000 }
gfCNCPoint1[10464] = {X 272.1770, Y 98.9257, Z -1.3333, A 0.000, B 0.000, C 0.000 }
gfCNCPoint1[10465] = {X 272.0727, Y 98.0000, Z -1.3333, A 0.000, B 0.000, C 0.000 }
gfCNCPoint1[10466] = {X 272.0727, Y 97.0659, Z -1.3333, A 0.000, B 0.000, C 0.000 }
gfCNCPoint1[10467] = {X 272.1633, Y 96.2022, Z -1.3333, A 0.000, B 0.000, C 0.000 }
gfCNCPoint1[10468] = {X 272.4314, Y 95.3761, Z -1.3333, A 0.000, B 0.000, C 0.000 }
gfCNCPoint1[10469] = {X 272.8650, Y 94.6237, Z -1.3333, A 0.000, B 0.000, C 0.000 }
gfCNCPoint1[10470] = {X 273.4455, Y 93.9777, Z -1.3333, A 0.000, B 0.000, C 0.000 }
gfCNCPoint1[10471] = {X 274.1474, Y 93.4663, Z -1.3333, A 0.000, B 0.000, C 0.000 }
gfCNCPoint1[10472] = {X 274.9402, Y 93.1118, Z -1.3333, A 0.000, B 0.000, C 0.000 }
gfCNCPoint1[10473] = {X 275.7894, Y 92.9296, Z -1.3333, A 0.000, B 0.000, C 0.000 }
gfCNCPoint1[10474] = {X 275.7894, Y 85.4858, Z -1.3333, A 0.000, B 0.000, C 0.000 }
gfCNCPoint1[10475] = {X 262.6227, Y 80.3245, Z -1.3333, A 0.000, B 0.000, C 0.000 }
gfCNCPoint1[10476] = {X 262.1894, Y 80.5969, Z -1.3333, A 0.000, B 0.000, C 0.000 }
gfCNCPoint1[10477] = {X 237.6349, Y 96.5014, Z -1.3333, A 0.000, B 0.000, C 0.000 }
gfCNCPoint1[10478] = {X 237.6398, Y 97.0652, Z -1.3333, A 0.000, B 0.000, C 0.000 }
gfCNCPoint1[10479] = {X 237.6398, Y 98.0000, Z -1.3333, A 0.000, B 0.000, C 0.000 }
gfCNCPoint1[10480] = {X 237.5355, Y 98.9257, Z -1.3333, A 0.000, B 0.000, C 0.000 }
gfCNCPoint1[10481] = {X 237.2278, Y 99.8050, Z -1.3333, A 0.000, B 0.000, C 0.000 }
gfCNCPoint1[10482] = {X 236.7322, Y 100.5937, Z -1.3333, A 0.000, B 0.000, C 0.000 }
gfCNCPoint1[10483] = {X 236.0735, Y 101.2524, Z -1.3333, A 0.000, B 0.000, C 0.000 }
gfCNCPoint1[10484] = {X 235.2847, Y 101.7480, Z -1.3333, A 0.000, B 0.000, C 0.000 }
gfCNCPoint1[10485] = {X 234.4055, Y 102.0557, Z -1.3333, A 0.000, B 0.000, C 0.000 }
gfCNCPoint1[10486] = {X 233.4798, Y 102.1600, Z -1.3333, A 0.000, B 0.000, C 0.000 }
gfCNCPoint1[10487] = {X 214.1790, Y 102.1600, Z -1.3333, A 0.000, B 0.000, C 0.000 }
gfCNCPoint1[10488] = {X 213.7860, Y 102.1414, Z -1.3333, A 0.000, B 0.000, C 0.000 }
gfCNCPoint1[10489] = {X 213.3966, Y 102.0857, Z -1.3333, A 0.000, B 0.000, C 0.000 }
gfCNCPoint1[10490] = {X 213.0071, Y 102.1414, Z -1.3333, A 0.000, B 0.000, C 0.000 }
gfCNCPoint1[10491] = {X 212.6141, Y 102.1600, Z -1.3333, A 0.000, B 0.000, C 0.000 }
gfCNCPoint1[10492] = {X 194.9870, Y 102.1600, Z -1.3333, A 0.000, B 0.000, C 0.000 }
gfCNCPoint1[10493] = {X 194.0613, Y 102.0557, Z -1.3333, A 0.000, B 0.000, C 0.000 }
gfCNCPoint1[10494] = {X 193.1820, Y 101.7480, Z -1.3333, A 0.000, B 0.000, C 0.000 }
gfCNCPoint1[10495] = {X 192.3932, Y 101.2524, Z -1.3333, A 0.000, B 0.000, C 0.000 }
gfCNCPoint1[10496] = {X 191.7345, Y 100.5937, Z -1.3333, A 0.000, B 0.000, C 0.000 }
gfCNCPoint1[10497] = {X 191.2389, Y 99.8050, Z -1.3333, A 0.000, B 0.000, C 0.000 }
gfCNCPoint1[10498] = {X 190.9313, Y 98.9257, Z -1.3333, A 0.000, B 0.000, C 0.000 }
gfCNCPoint1[10499] = {X 190.8270, Y 98.0000, Z -1.3333, A 0.000, B 0.000, C 0.000 }
gfCNCPoint1[10500] = {X 190.8270, Y 97.0659, Z -1.3333, A 0.000, B 0.000, C 0.000 }
gfCNCPoint1[10501] = {X 190.9241, Y 96.1723, Z -1.3333, A 0.000, B 0.000, C 0.000 }
gfCNCPoint1[10502] = {X 191.2109, Y 95.3203, Z -1.3333, A 0.000, B 0.000, C 0.000 }
gfCNCPoint1[10503] = {X 191.6741, Y 94.5499, Z -1.3333, A 0.000, B 0.000, C 0.000 }
gfCNCPoint1[10504] = {X 191.7354, Y 94.4712, Z -1.3333, A 0.000, B 0.000, C 0.000 }
gfCNCPoint1[10505] = {X 191.7986, Y 94.3939, Z -1.3333, A 0.000, B 0.000, C 0.000 }
gfCNCPoint1[10506] = {X 188.6351, Y 90.9402, Z -1.3333, A 0.000, B 0.000, C 0.000 }
gfCNCPoint1[10507] = {X 150.0187, Y 90.9402, Z -1.3333, A 0.000, B 0.000, C 0.000 }
gfCNCPoint1[10508] = {X 146.9329, Y 94.3590, Z -1.3333, A 0.000, B 0.000, C 0.000 }
gfCNCPoint1[10509] = {X 147.4786, Y 95.1734, Z -1.3333, A 0.000, B 0.000, C 0.000 }
gfCNCPoint1[10510] = {X 147.8202, Y 96.0923, Z -1.3333, A 0.000, B 0.000, C 0.000 }
gfCNCPoint1[10511] = {X 147.9391, Y 97.0654, Z -1.3333, A 0.000, B 0.000, C 0.000 }
gfCNCPoint1[10512] = {X 147.9391, Y 98.0000, Z -1.3333, A 0.000, B 0.000, C 0.000 }
gfCNCPoint1[10513] = {X 147.8348, Y 98.9257, Z -1.3333, A 0.000, B 0.000, C 0.000 }
gfCNCPoint1[10514] = {X 147.5271, Y 99.8050, Z -1.3333, A 0.000, B 0.000, C 0.000 }
gfCNCPoint1[10515] = {X 147.0315, Y 100.5937, Z -1.3333, A 0.000, B 0.000, C 0.000 }
gfCNCPoint1[10516] = {X 146.3728, Y 101.2524, Z -1.3333, A 0.000, B 0.000, C 0.000 }
gfCNCPoint1[10517] = {X 145.5841, Y 101.7480, Z -1.3333, A 0.000, B 0.000, C 0.000 }
gfCNCPoint1[10518] = {X 144.7048, Y 102.0557, Z -1.3333, A 0.000, B 0.000, C 0.000 }
gfCNCPoint1[10519] = {X 143.7791, Y 102.1600, Z -1.3333, A 0.000, B 0.000, C 0.000 }
gfCNCPoint1[10520] = {X 125.0000, Y 102.1600, Z -1.3333, A 0.000, B 0.000, C 0.000 }
gfCNCPoint1[10521] = {X 124.0743, Y 102.0557, Z -1.3333, A 0.000, B 0.000, C 0.000 }
gfCNCPoint1[10522] = {X 123.1950, Y 101.7480, Z -1.3333, A 0.000, B 0.000, C 0.000 }
gfCNCPoint1[10523] = {X 122.4063, Y 101.2524, Z -1.3333, A 0.000, B 0.000, C 0.000 }
gfCNCPoint1[10524] = {X 121.7476, Y 100.5937, Z -1.3333, A 0.000, B 0.000, C 0.000 }
gfCNCPoint1[10525] = {X 121.2520, Y 99.8050, Z -1.3333, A 0.000, B 0.000, C 0.000 }
gfCNCPoint1[10526] = {X 120.9443, Y 98.9257, Z -1.3333, A 0.000, B 0.000, C 0.000 }
gfCNCPoint1[10527] = {X 120.8400, Y 98.0000, Z -1.3333, A 0.000, B 0.000, C 0.000 }
gfCNCPoint1[10528] = {X 120.8400, Y 97.0659, Z -1.3333, A 0.000, B 0.000, C 0.000 }
gfCNCPoint1[10529] = {X 120.9406, Y 96.1564, Z -1.3333, A 0.000, B 0.000, C 0.000 }
gfCNCPoint1[10530] = {X 121.2377, Y 95.2909, Z -1.3333, A 0.000, B 0.000, C 0.000 }
gfCNCPoint1[10531] = {X 121.7168, Y 94.5113, Z -1.3333, A 0.000, B 0.000, C 0.000 }
gfCNCPoint1[10532] = {X 122.3548, Y 93.8552, Z -1.3333, A 0.000, B 0.000, C 0.000 }
gfCNCPoint1[10533] = {X 123.1208, Y 93.3546, Z -1.3333, A 0.000, B 0.000, C 0.000 }
gfCNCPoint1[10534] = {X 123.9777, Y 93.0335, Z -1.3333, A 0.000, B 0.000, C 0.000 }
gfCNCPoint1[10535] = {X 124.8840, Y 92.9076, Z -1.3333, A 0.000, B 0.000, C 0.000 }
gfCNCPoint1[10536] = {X 124.9163, Y 92.8904, Z -1.3333, A 0.000, B 0.000, C 0.000 }
gfCNCPoint1[10537] = {X 124.9515, Y 92.8811, Z -1.3333, A 0.000, B 0.000, C 0.000 }
gfCNCPoint1[10538] = {X 125.4721, Y 92.8038, Z -1.3333, A 0.000, B 0.000, C 0.000 }
gfCNCPoint1[10539] = {X 126.3318, Y 92.6575, Z -1.3333, A 0.000, B 0.000, C 0.000 }
gfCNCPoint1[10540] = {X 127.1796, Y 92.4531, Z -1.3333, A 0.000, B 0.000, C 0.000 }
gfCNCPoint1[10541] = {X 128.4223, Y 91.2833, Z -1.3333, A 0.000, B 0.000, C 0.000 }
gfCNCPoint1[10542] = {X 129.5991, Y 90.0473, Z -1.3333, A 0.000, B 0.000, C 0.000 }
gfCNCPoint1[10543] = {X 140.7989, Y 77.7485, Z -1.3333, A 0.000, B 0.000, C 0.000 }
gfCNCPoint1[10544] = {X 137.8414, Y 75.0553, Z -1.3333, A 0.000, B 0.000, C 0.000 }
gfCNCPoint1[10545] = {X 140.8580, Y 77.8024, Z -1.3333, A 0.000, B 0.000, C 0.000 }
gfCNCPoint1[10546] = {X 155.9356, Y 61.2452, Z -1.3333, A 0.000, B 0.000, C 0.000 }
gfCNCPoint1[10547] = {X 155.5468, Y 60.5387, Z -1.3333, A 0.000, B 0.000, C 0.000 }
gfCNCPoint1[10548] = {X 155.3044, Y 59.7696, Z -1.3333, A 0.000, B 0.000, C 0.000 }
gfCNCPoint1[10549] = {X 155.2181, Y 58.9678, Z -1.3333, A 0.000, B 0.000, C 0.000 }
gfCNCPoint1[10550] = {X 155.2180, Y 58.0000, Z -1.3333, A 0.000, B 0.000, C 0.000 }
gfCNCPoint1[10551] = {X 155.3203, Y 57.0921, Z -1.3333, A 0.000, B 0.000, C 0.000 }
gfCNCPoint1[10552] = {X 155.6220, Y 56.2298, Z -1.3333, A 0.000, B 0.000, C 0.000 }
gfCNCPoint1[10553] = {X 156.1081, Y 55.4562, Z -1.3333, A 0.000, B 0.000, C 0.000 }
gfCNCPoint1[10554] = {X 156.7541, Y 54.8101, Z -1.3333, A 0.000, B 0.000, C 0.000 }
gfCNCPoint1[10555] = {X 157.5277, Y 54.3240, Z -1.3333, A 0.000, B 0.000, C 0.000 }
gfCNCPoint1[10556] = {X 158.3901, Y 54.0223, Z -1.3333, A 0.000, B 0.000, C 0.000 }
gfCNCPoint1[10557] = {X 159.2980, Y 53.9200, Z -1.3333, A 0.000, B 0.000, C 0.000 }
gfCNCPoint1[10558] = {X 178.5335, Y 53.9200, Z -1.3333, A 0.000, B 0.000, C 0.000 }
gfCNCPoint1[10559] = {X 179.4414, Y 54.0223, Z -1.3333, A 0.000, B 0.000, C 0.000 }
gfCNCPoint1[10560] = {X 180.3037, Y 54.3240, Z -1.3333, A 0.000, B 0.000, C 0.000 }
gfCNCPoint1[10561] = {X 181.0773, Y 54.8101, Z -1.3333, A 0.000, B 0.000, C 0.000 }
gfCNCPoint1[10562] = {X 181.7234, Y 55.4562, Z -1.3333, A 0.000, B 0.000, C 0.000 }
gfCNCPoint1[10563] = {X 182.2095, Y 56.2298, Z -1.3333, A 0.000, B 0.000, C 0.000 }
gfCNCPoint1[10564] = {X 182.5112, Y 57.0921, Z -1.3333, A 0.000, B 0.000, C 0.000 }
gfCNCPoint1[10565] = {X 182.6135, Y 58.0000, Z -1.3333, A 0.000, B 0.000, C 0.000 }
gfCNCPoint1[10566] = {X 182.6135, Y 58.9342, Z -1.3333, A 0.000, B 0.000, C 0.000 }
gfCNCPoint1[10567] = {X 182.5334, Y 59.7387, Z -1.3333, A 0.000, B 0.000, C 0.000 }
gfCNCPoint1[10568] = {X 182.2962, Y 60.5116, Z -1.3333, A 0.000, B 0.000, C 0.000 }
gfCNCPoint1[10569] = {X 181.9113, Y 61.2225, Z -1.3333, A 0.000, B 0.000, C 0.000 }
gfCNCPoint1[10570] = {X 209.3002, Y 91.1159, Z -1.3333, A 0.000, B 0.000, C 0.000 }
gfCNCPoint1[10571] = {X 209.9709, Y 91.7964, Z -1.3333, A 0.000, B 0.000, C 0.000 }
gfCNCPoint1[10572] = {X 210.6894, Y 92.4263, Z -1.3333, A 0.000, B 0.000, C 0.000 }
gfCNCPoint1[10573] = {X 211.0143, Y 92.6313, Z -1.3333, A 0.000, B 0.000, C 0.000 }
gfCNCPoint1[10574] = {X 211.3787, Y 92.7529, Z -1.3333, A 0.000, B 0.000, C 0.000 }
gfCNCPoint1[10575] = {X 212.3974, Y 92.9413, Z -1.3333, A 0.000, B 0.000, C 0.000 }
gfCNCPoint1[10576] = {X 213.4269, Y 93.0569, Z -1.3333, A 0.000, B 0.000, C 0.000 }
gfCNCPoint1[10577] = {X 214.4700, Y 92.9772, Z -1.3333, A 0.000, B 0.000, C 0.000 }
gfCNCPoint1[10578] = {X 215.5143, Y 92.9168, Z -1.3333, A 0.000, B 0.000, C 0.000 }
gfCNCPoint1[10579] = {X 216.2274, Y 92.8383, Z -1.3333, A 0.000, B 0.000, C 0.000 }
gfCNCPoint1[10580] = {X 216.9141, Y 92.6303, Z -1.3333, A 0.000, B 0.000, C 0.000 }
gfCNCPoint1[10581] = {X 217.5511, Y 92.3001, Z -1.3333, A 0.000, B 0.000, C 0.000 }
gfCNCPoint1[10582] = {X 223.0910, Y 88.7249, Z -1.3333, A 0.000, B 0.000, C 0.000 }
gfCNCPoint1[10583] = {X 246.3554, Y 73.8480, Z -1.3333, A 0.000, B 0.000, C 0.000 }
gfCNCPoint1[10584] = {X 221.7196, Y 64.1795, Z -1.3333, A 0.000, B 0.000, C 0.000 }
gfCNCPoint1[10585] = {X 219.9262, Y 63.5792, Z -1.3333, A 0.000, B 0.000, C 0.000 }
gfCNCPoint1[10586] = {X 218.0759, Y 63.1883, Z -1.3333, A 0.000, B 0.000, C 0.000 }
gfCNCPoint1[10587] = {X 216.1929, Y 63.0117, Z -1.3333, A 0.000, B 0.000, C 0.000 }
gfCNCPoint1[10588] = {X 215.3127, Y 62.8850, Z -1.3333, A 0.000, B 0.000, C 0.000 }
gfCNCPoint1[10589] = {X 214.4809, Y 62.5706, Z -1.3333, A 0.000, B 0.000, C 0.000 }
gfCNCPoint1[10590] = {X 213.7370, Y 62.0834, Z -1.3333, A 0.000, B 0.000, C 0.000 }
gfCNCPoint1[10591] = {X 213.1162, Y 61.4466, Z -1.3333, A 0.000, B 0.000, C 0.000 }
gfCNCPoint1[10592] = {X 212.6482, Y 60.6905, Z -1.3333, A 0.000, B 0.000, C 0.000 }
gfCNCPoint1[10593] = {X 212.3552, Y 59.8509, Z -1.3333, A 0.000, B 0.000, C 0.000 }
gfCNCPoint1[10594] = {X 212.2509, Y 58.9678, Z -1.3333, A 0.000, B 0.000, C 0.000 }
gfCNCPoint1[10595] = {X 212.2508, Y 58.0000, Z -1.3333, A 0.000, B 0.000, C 0.000 }
gfCNCPoint1[10596] = {X 212.3531, Y 57.0921, Z -1.3333, A 0.000, B 0.000, C 0.000 }
gfCNCPoint1[10597] = {X 212.6549, Y 56.2298, Z -1.3333, A 0.000, B 0.000, C 0.000 }
gfCNCPoint1[10598] = {X 213.1409, Y 55.4562, Z -1.3333, A 0.000, B 0.000, C 0.000 }
gfCNCPoint1[10599] = {X 213.7870, Y 54.8101, Z -1.3333, A 0.000, B 0.000, C 0.000 }
gfCNCPoint1[10600] = {X 214.5606, Y 54.3240, Z -1.3333, A 0.000, B 0.000, C 0.000 }
gfCNCPoint1[10601] = {X 215.4229, Y 54.0223, Z -1.3333, A 0.000, B 0.000, C 0.000 }
gfCNCPoint1[10602] = {X 216.3308, Y 53.9200, Z -1.3333, A 0.000, B 0.000, C 0.000 }
gfCNCPoint1[10603] = {X 237.2617, Y 53.9200, Z -1.3333, A 0.000, B 0.000, C 0.000 }
gfCNCPoint1[10604] = {X 238.1696, Y 54.0223, Z -1.3333, A 0.000, B 0.000, C 0.000 }
gfCNCPoint1[10605] = {X 239.0319, Y 54.3240, Z -1.3333, A 0.000, B 0.000, C 0.000 }
gfCNCPoint1[10606] = {X 239.8055, Y 54.8101, Z -1.3333, A 0.000, B 0.000, C 0.000 }
gfCNCPoint1[10607] = {X 240.4516, Y 55.4562, Z -1.3333, A 0.000, B 0.000, C 0.000 }
gfCNCPoint1[10608] = {X 240.9376, Y 56.2298, Z -1.3333, A 0.000, B 0.000, C 0.000 }
gfCNCPoint1[10609] = {X 241.2394, Y 57.0921, Z -1.3333, A 0.000, B 0.000, C 0.000 }
gfCNCPoint1[10610] = {X 241.3417, Y 58.0000, Z -1.3333, A 0.000, B 0.000, C 0.000 }
gfCNCPoint1[10611] = {X 241.3417, Y 58.3971, Z -1.3333, A 0.000, B 0.000, C 0.000 }
gfCNCPoint1[10612] = {X 248.0246, Y 61.0026, Z -1.3333, A 0.000, B 0.000, C 0.000 }
gfCNCPoint1[10613] = {X 275.8741, Y 72.0566, Z -1.3333, A 0.000, B 0.000, C 0.000 }
gfCNCPoint1[10614] = {X 275.8746, Y 62.9983, Z -1.3333, A 0.000, B 0.000, C 0.000 }
gfCNCPoint1[10615] = {X 275.7384, Y 62.9840, Z -1.3333, A 0.000, B 0.000, C 0.000 }
gfCNCPoint1[10616] = {X 275.6027, Y 62.9651, Z -1.3333, A 0.000, B 0.000, C 0.000 }
gfCNCPoint1[10617] = {X 274.6830, Y 62.7083, Z -1.3333, A 0.000, B 0.000, C 0.000 }
gfCNCPoint1[10618] = {X 273.8481, Y 62.2447, Z -1.3333, A 0.000, B 0.000, C 0.000 }
gfCNCPoint1[10619] = {X 273.1439, Y 61.5998, Z -1.3333, A 0.000, B 0.000, C 0.000 }
gfCNCPoint1[10620] = {X 272.6089, Y 60.8088, Z -1.3333, A 0.000, B 0.000, C 0.000 }
gfCNCPoint1[10621] = {X 272.2724, Y 59.9152, Z -1.3333, A 0.000, B 0.000, C 0.000 }
gfCNCPoint1[10622] = {X 272.1528, Y 58.9678, Z -1.3333, A 0.000, B 0.000, C 0.000 }
gfCNCPoint1[10623] = {X 272.1527, Y 58.0000, Z -1.3333, A 0.000, B 0.000, C 0.000 }
gfCNCPoint1[10624] = {X 272.2550, Y 57.0921, Z -1.3333, A 0.000, B 0.000, C 0.000 }
gfCNCPoint1[10625] = {X 272.5567, Y 56.2298, Z -1.3333, A 0.000, B 0.000, C 0.000 }
gfCNCPoint1[10626] = {X 273.0428, Y 55.4562, Z -1.3333, A 0.000, B 0.000, C 0.000 }
gfCNCPoint1[10627] = {X 273.6889, Y 54.8101, Z -1.3333, A 0.000, B 0.000, C 0.000 }
gfCNCPoint1[10628] = {X 274.4624, Y 54.3240, Z -1.3333, A 0.000, B 0.000, C 0.000 }
gfCNCPoint1[10629] = {X 275.3248, Y 54.0223, Z -1.3333, A 0.000, B 0.000, C 0.000 }
gfCNCPoint1[10630] = {X 276.2327, Y 53.9200, Z -1.3333, A 0.000, B 0.000, C 0.000 }
gfCNCPoint1[10631] = {X 292.7731, Y 53.9200, Z -1.3333, A 0.000, B 0.000, C 0.000 }
gfCNCPoint1[10632] = {X 293.6810, Y 54.0223, Z -1.3333, A 0.000, B 0.000, C 0.000 }
gfCNCPoint1[10633] = {X 294.5433, Y 54.3240, Z -1.3333, A 0.000, B 0.000, C 0.000 }
gfCNCPoint1[10634] = {X 295.3169, Y 54.8101, Z -1.3333, A 0.000, B 0.000, C 0.000 }
gfCNCPoint1[10635] = {X 295.9630, Y 55.4562, Z -1.3333, A 0.000, B 0.000, C 0.000 }
gfCNCPoint1[10636] = {X 296.4490, Y 56.2298, Z -1.3333, A 0.000, B 0.000, C 0.000 }
gfCNCPoint1[10637] = {X 296.7508, Y 57.0921, Z -1.3333, A 0.000, B 0.000, C 0.000 }
gfCNCPoint1[10638] = {X 296.8531, Y 58.0000, Z -1.3333, A 0.000, B 0.000, C 0.000 }
gfCNCPoint1[10639] = {X 296.8531, Y 58.9344, Z -1.3333, A 0.000, B 0.000, C 0.000 }
gfCNCPoint1[10640] = {X 296.7372, Y 59.8874, Z -1.3333, A 0.000, B 0.000, C 0.000 }
gfCNCPoint1[10641] = {X 296.4027, Y 60.7872, Z -1.3333, A 0.000, B 0.000, C 0.000 }
gfCNCPoint1[10642] = {X 295.8681, Y 61.5846, Z -1.3333, A 0.000, B 0.000, C 0.000 }
gfCNCPoint1[10643] = {X 295.1625, Y 62.2356, Z -1.3333, A 0.000, B 0.000, C 0.000 }
gfCNCPoint1[10644] = {X 294.3249, Y 62.7045, Z -1.3333, A 0.000, B 0.000, C 0.000 }
gfCNCPoint1[10645] = {X 293.4011, Y 62.9657, Z -1.3333, A 0.000, B 0.000, C 0.000 }
gfCNCPoint1[10646] = {X 293.2748, Y 62.9838, Z -1.3333, A 0.000, B 0.000, C 0.000 }
gfCNCPoint1[10647] = {X 293.1480, Y 62.9980, Z -1.3333, A 0.000, B 0.000, C 0.000 }
gfCNCPoint1[10648] = {X 293.1314, Y 63.1582, Z -1.3333, A 0.000, B 0.000, C 0.000 }
gfCNCPoint1[10649] = {X 293.1441, Y 92.9944, Z -1.3333, A 0.000, B 0.000, C 0.000 }
gfCNCPoint1[10650] = {X 293.2723, Y 93.0091, Z -1.3333, A 0.000, B 0.000, C 0.000 }
gfCNCPoint1[10651] = {X 293.4001, Y 93.0278, Z -1.3333, A 0.000, B 0.000, C 0.000 }
gfCNCPoint1[10652] = {X 294.3236, Y 93.2916, Z -1.3333, A 0.000, B 0.000, C 0.000 }
gfCNCPoint1[10653] = {X 295.1608, Y 93.7623, Z -1.3333, A 0.000, B 0.000, C 0.000 }
gfCNCPoint1[10654] = {X 295.8660, Y 94.4144, Z -1.3333, A 0.000, B 0.000, C 0.000 }
gfCNCPoint1[10655] = {X 296.4007, Y 95.2123, Z -1.3333, A 0.000, B 0.000, C 0.000 }
gfCNCPoint1[10656] = {X 296.7359, Y 96.1124, Z -1.3333, A 0.000, B 0.000, C 0.000 }
gfCNCPoint1[10657] = {X 296.8531, Y 97.0657, Z -1.3333, A 0.000, B 0.000, C 0.000 }
gfCNCPoint1[10658] = {X 296.8531, Y 98.0000, Z -1.3333, A 0.000, B 0.000, C 0.000 }
gfCNCPoint1[10659] = {X 296.7508, Y 98.9079, Z -1.3333, A 0.000, B 0.000, C 0.000 }
gfCNCPoint1[10660] = {X 296.4490, Y 99.7702, Z -1.3333, A 0.000, B 0.000, C 0.000 }
gfCNCPoint1[10661] = {X 295.9630, Y 100.5438, Z -1.3333, A 0.000, B 0.000, C 0.000 }
gfCNCPoint1[10662] = {X 295.3169, Y 101.1899, Z -1.3333, A 0.000, B 0.000, C 0.000 }
gfCNCPoint1[10663] = {X 294.5433, Y 101.6760, Z -1.3333, A 0.000, B 0.000, C 0.000 }
gfCNCPoint1[10664] = {X 293.6810, Y 101.9777, Z -1.3333, A 0.000, B 0.000, C 0.000 }
gfCNCPoint1[10665] = {X 292.7731, Y 102.0800, Z -1.3333, A 0.000, B 0.000, C 0.000 }
gfCNCPoint1[10666] = {X 276.2327, Y 102.0800, Z -1.3333, A 0.000, B 0.000, C 0.000 }
gfCNCPoint1[10667] = {X 275.3248, Y 101.9777, Z -1.3333, A 0.000, B 0.000, C 0.000 }
gfCNCPoint1[10668] = {X 274.4624, Y 101.6760, Z -1.3333, A 0.000, B 0.000, C 0.000 }
gfCNCPoint1[10669] = {X 273.6889, Y 101.1899, Z -1.3333, A 0.000, B 0.000, C 0.000 }
gfCNCPoint1[10670] = {X 273.0428, Y 100.5438, Z -1.3333, A 0.000, B 0.000, C 0.000 }
gfCNCPoint1[10671] = {X 272.5567, Y 99.7702, Z -1.3333, A 0.000, B 0.000, C 0.000 }
gfCNCPoint1[10672] = {X 272.2550, Y 98.9079, Z -1.3333, A 0.000, B 0.000, C 0.000 }
gfCNCPoint1[10673] = {X 272.1527, Y 98.0000, Z -1.3333, A 0.000, B 0.000, C 0.000 }
gfCNCPoint1[10674] = {X 272.1527, Y 97.0659, Z -1.3333, A 0.000, B 0.000, C 0.000 }
gfCNCPoint1[10675] = {X 272.2437, Y 96.2088, Z -1.3333, A 0.000, B 0.000, C 0.000 }
gfCNCPoint1[10676] = {X 272.5128, Y 95.3899, Z -1.3333, A 0.000, B 0.000, C 0.000 }
gfCNCPoint1[10677] = {X 272.9480, Y 94.6458, Z -1.3333, A 0.000, B 0.000, C 0.000 }
gfCNCPoint1[10678] = {X 273.5297, Y 94.0098, Z -1.3333, A 0.000, B 0.000, C 0.000 }
gfCNCPoint1[10679] = {X 274.2321, Y 93.5101, Z -1.3333, A 0.000, B 0.000, C 0.000 }
gfCNCPoint1[10680] = {X 275.0238, Y 93.1692, Z -1.3333, A 0.000, B 0.000, C 0.000 }
gfCNCPoint1[10681] = {X 275.8694, Y 93.0021, Z -1.3333, A 0.000, B 0.000, C 0.000 }
gfCNCPoint1[10682] = {X 275.8694, Y 85.4313, Z -1.3333, A 0.000, B 0.000, C 0.000 }
gfCNCPoint1[10683] = {X 262.6143, Y 80.2352, Z -1.3333, A 0.000, B 0.000, C 0.000 }
gfCNCPoint1[10684] = {X 262.1464, Y 80.5294, Z -1.3333, A 0.000, B 0.000, C 0.000 }
gfCNCPoint1[10685] = {X 237.5546, Y 96.4581, Z -1.3333, A 0.000, B 0.000, C 0.000 }
gfCNCPoint1[10686] = {X 237.5598, Y 97.0656, Z -1.3333, A 0.000, B 0.000, C 0.000 }
gfCNCPoint1[10687] = {X 237.5598, Y 98.0000, Z -1.3333, A 0.000, B 0.000, C 0.000 }
gfCNCPoint1[10688] = {X 237.4575, Y 98.9079, Z -1.3333, A 0.000, B 0.000, C 0.000 }
gfCNCPoint1[10689] = {X 237.1557, Y 99.7702, Z -1.3333, A 0.000, B 0.000, C 0.000 }
gfCNCPoint1[10690] = {X 236.6697, Y 100.5438, Z -1.3333, A 0.000, B 0.000, C 0.000 }
gfCNCPoint1[10691] = {X 236.0236, Y 101.1899, Z -1.3333, A 0.000, B 0.000, C 0.000 }
gfCNCPoint1[10692] = {X 235.2500, Y 101.6760, Z -1.3333, A 0.000, B 0.000, C 0.000 }
gfCNCPoint1[10693] = {X 234.3877, Y 101.9777, Z -1.3333, A 0.000, B 0.000, C 0.000 }
gfCNCPoint1[10694] = {X 233.4798, Y 102.0800, Z -1.3333, A 0.000, B 0.000, C 0.000 }
gfCNCPoint1[10695] = {X 214.1790, Y 102.0800, Z -1.3333, A 0.000, B 0.000, C 0.000 }
gfCNCPoint1[10696] = {X 213.7860, Y 102.0610, Z -1.3333, A 0.000, B 0.000, C 0.000 }
gfCNCPoint1[10697] = {X 213.3966, Y 102.0043, Z -1.3333, A 0.000, B 0.000, C 0.000 }
gfCNCPoint1[10698] = {X 213.0072, Y 102.0610, Z -1.3333, A 0.000, B 0.000, C 0.000 }
gfCNCPoint1[10699] = {X 212.6141, Y 102.0800, Z -1.3333, A 0.000, B 0.000, C 0.000 }
gfCNCPoint1[10700] = {X 194.9870, Y 102.0800, Z -1.3333, A 0.000, B 0.000, C 0.000 }
gfCNCPoint1[10701] = {X 194.0791, Y 101.9777, Z -1.3333, A 0.000, B 0.000, C 0.000 }
gfCNCPoint1[10702] = {X 193.2167, Y 101.6760, Z -1.3333, A 0.000, B 0.000, C 0.000 }
gfCNCPoint1[10703] = {X 192.4431, Y 101.1899, Z -1.3333, A 0.000, B 0.000, C 0.000 }
gfCNCPoint1[10704] = {X 191.7971, Y 100.5438, Z -1.3333, A 0.000, B 0.000, C 0.000 }
gfCNCPoint1[10705] = {X 191.3110, Y 99.7702, Z -1.3333, A 0.000, B 0.000, C 0.000 }
gfCNCPoint1[10706] = {X 191.0093, Y 98.9079, Z -1.3333, A 0.000, B 0.000, C 0.000 }
gfCNCPoint1[10707] = {X 190.9070, Y 98.0000, Z -1.3333, A 0.000, B 0.000, C 0.000 }
gfCNCPoint1[10708] = {X 190.9070, Y 97.0659, Z -1.3333, A 0.000, B 0.000, C 0.000 }
gfCNCPoint1[10709] = {X 191.0022, Y 96.1894, Z -1.3333, A 0.000, B 0.000, C 0.000 }
gfCNCPoint1[10710] = {X 191.2835, Y 95.3539, Z -1.3333, A 0.000, B 0.000, C 0.000 }
gfCNCPoint1[10711] = {X 191.7378, Y 94.5983, Z -1.3333, A 0.000, B 0.000, C 0.000 }
gfCNCPoint1[10712] = {X 191.8199, Y 94.4938, Z -1.3333, A 0.000, B 0.000, C 0.000 }
gfCNCPoint1[10713] = {X 191.9053, Y 94.3920, Z -1.3333, A 0.000, B 0.000, C 0.000 }
gfCNCPoint1[10714] = {X 188.6703, Y 90.8602, Z -1.3333, A 0.000, B 0.000, C 0.000 }
gfCNCPoint1[10715] = {X 149.9831, Y 90.8602, Z -1.3333, A 0.000, B 0.000, C 0.000 }
gfCNCPoint1[10716] = {X 146.8260, Y 94.3580, Z -1.3333, A 0.000, B 0.000, C 0.000 }
gfCNCPoint1[10717] = {X 147.3858, Y 95.1683, Z -1.3333, A 0.000, B 0.000, C 0.000 }
gfCNCPoint1[10718] = {X 147.7369, Y 96.0885, Z -1.3333, A 0.000, B 0.000, C 0.000 }
gfCNCPoint1[10719] = {X 147.8591, Y 97.0658, Z -1.3333, A 0.000, B 0.000, C 0.000 }
gfCNCPoint1[10720] = {X 147.8591, Y 98.0000, Z -1.3333, A 0.000, B 0.000, C 0.000 }
gfCNCPoint1[10721] = {X 147.7568, Y 98.9079, Z -1.3333, A 0.000, B 0.000, C 0.000 }
gfCNCPoint1[10722] = {X 147.4551, Y 99.7702, Z -1.3333, A 0.000, B 0.000, C 0.000 }
gfCNCPoint1[10723] = {X 146.9690, Y 100.5438, Z -1.3333, A 0.000, B 0.000, C 0.000 }
gfCNCPoint1[10724] = {X 146.3229, Y 101.1899, Z -1.3333, A 0.000, B 0.000, C 0.000 }
gfCNCPoint1[10725] = {X 145.5494, Y 101.6760, Z -1.3333, A 0.000, B 0.000, C 0.000 }
gfCNCPoint1[10726] = {X 144.6870, Y 101.9777, Z -1.3333, A 0.000, B 0.000, C 0.000 }
gfCNCPoint1[10727] = {X 143.7791, Y 102.0800, Z -1.3333, A 0.000, B 0.000, C 0.000 }
gfCNCPoint1[10728] = {X 125.0000, Y 102.0800, Z -1.3333, A 0.000, B 0.000, C 0.000 }
gfCNCPoint1[10729] = {X 124.0921, Y 101.9777, Z -1.3333, A 0.000, B 0.000, C 0.000 }
gfCNCPoint1[10730] = {X 123.2298, Y 101.6760, Z -1.3333, A 0.000, B 0.000, C 0.000 }
gfCNCPoint1[10731] = {X 122.4562, Y 101.1899, Z -1.3333, A 0.000, B 0.000, C 0.000 }
gfCNCPoint1[10732] = {X 121.8101, Y 100.5438, Z -1.3333, A 0.000, B 0.000, C 0.000 }
gfCNCPoint1[10733] = {X 121.3240, Y 99.7702, Z -1.3333, A 0.000, B 0.000, C 0.000 }
gfCNCPoint1[10734] = {X 121.0223, Y 98.9079, Z -1.3333, A 0.000, B 0.000, C 0.000 }
gfCNCPoint1[10735] = {X 120.9200, Y 98.0000, Z -1.3333, A 0.000, B 0.000, C 0.000 }
gfCNCPoint1[10736] = {X 120.9200, Y 97.0659, Z -1.3333, A 0.000, B 0.000, C 0.000 }
gfCNCPoint1[10737] = {X 121.0194, Y 96.1708, Z -1.3333, A 0.000, B 0.000, C 0.000 }
gfCNCPoint1[10738] = {X 121.3127, Y 95.3194, Z -1.3333, A 0.000, B 0.000, C 0.000 }
gfCNCPoint1[10739] = {X 121.7857, Y 94.5530, Z -1.3333, A 0.000, B 0.000, C 0.000 }
gfCNCPoint1[10740] = {X 122.4153, Y 93.9090, Z -1.3333, A 0.000, B 0.000, C 0.000 }
gfCNCPoint1[10741] = {X 123.1709, Y 93.4189, Z -1.3333, A 0.000, B 0.000, C 0.000 }
gfCNCPoint1[10742] = {X 124.0155, Y 93.1065, Z -1.3333, A 0.000, B 0.000, C 0.000 }
gfCNCPoint1[10743] = {X 124.9082, Y 92.9870, Z -1.3333, A 0.000, B 0.000, C 0.000 }
gfCNCPoint1[10744] = {X 124.9322, Y 92.9717, Z -1.3333, A 0.000, B 0.000, C 0.000 }
gfCNCPoint1[10745] = {X 124.9633, Y 92.9602, Z -1.3333, A 0.000, B 0.000, C 0.000 }
gfCNCPoint1[10746] = {X 125.4828, Y 92.8831, Z -1.3333, A 0.000, B 0.000, C 0.000 }
gfCNCPoint1[10747] = {X 126.3570, Y 92.7340, Z -1.3333, A 0.000, B 0.000, C 0.000 }
gfCNCPoint1[10748] = {X 127.2189, Y 92.5252, Z -1.3333, A 0.000, B 0.000, C 0.000 }
gfCNCPoint1[10749] = {X 128.4721, Y 91.3466, Z -1.3333, A 0.000, B 0.000, C 0.000 }
gfCNCPoint1[10750] = {X 129.6586, Y 90.1009, Z -1.3333, A 0.000, B 0.000, C 0.000 }
gfCNCPoint1[10751] = {X 140.8580, Y 77.8024, Z -1.3333, A 0.000, B 0.000, C 0.000 }
gfCNCPoint1[10752] = {X 137.8979, Y 75.1068, Z -1.3333, A 0.000, B 0.000, C 0.000 }
gfCNCPoint1[10753] = {X 137.8983, Y 75.1063, Z -1.3333, A 0.000, B 0.000, C 0.000 }
gfCNCPoint1[10754] = {X 140.9145, Y 77.8539, Z -1.3333, A 0.000, B 0.000, C 0.000 }
gfCNCPoint1[10755] = {X 156.0378, Y 61.2518, Z -1.3333, A 0.000, B 0.000, C 0.000 }
gfCNCPoint1[10756] = {X 155.6327, Y 60.5359, Z -1.3333, A 0.000, B 0.000, C 0.000 }
gfCNCPoint1[10757] = {X 155.3825, Y 59.7523, Z -1.3333, A 0.000, B 0.000, C 0.000 }
gfCNCPoint1[10758] = {X 155.2980, Y 58.9340, Z -1.3333, A 0.000, B 0.000, C 0.000 }
gfCNCPoint1[10759] = {X 155.2980, Y 58.0000, Z -1.3333, A 0.000, B 0.000, C 0.000 }
gfCNCPoint1[10760] = {X 155.3982, Y 57.1099, Z -1.3333, A 0.000, B 0.000, C 0.000 }
gfCNCPoint1[10761] = {X 155.6941, Y 56.2645, Z -1.3333, A 0.000, B 0.000, C 0.000 }
gfCNCPoint1[10762] = {X 156.1706, Y 55.5060, Z -1.3333, A 0.000, B 0.000, C 0.000 }
gfCNCPoint1[10763] = {X 156.8040, Y 54.8727, Z -1.3333, A 0.000, B 0.000, C 0.000 }
gfCNCPoint1[10764] = {X 157.5624, Y 54.3961, Z -1.3333, A 0.000, B 0.000, C 0.000 }
gfCNCPoint1[10765] = {X 158.4079, Y 54.1003, Z -1.3333, A 0.000, B 0.000, C 0.000 }
gfCNCPoint1[10766] = {X 159.2980, Y 54.0000, Z -1.3333, A 0.000, B 0.000, C 0.000 }
gfCNCPoint1[10767] = {X 178.5335, Y 54.0000, Z -1.3333, A 0.000, B 0.000, C 0.000 }
gfCNCPoint1[10768] = {X 179.4236, Y 54.1003, Z -1.3333, A 0.000, B 0.000, C 0.000 }
gfCNCPoint1[10769] = {X 180.2690, Y 54.3961, Z -1.3333, A 0.000, B 0.000, C 0.000 }
gfCNCPoint1[10770] = {X 181.0275, Y 54.8727, Z -1.3333, A 0.000, B 0.000, C 0.000 }
gfCNCPoint1[10771] = {X 181.6608, Y 55.5060, Z -1.3333, A 0.000, B 0.000, C 0.000 }
gfCNCPoint1[10772] = {X 182.1374, Y 56.2645, Z -1.3333, A 0.000, B 0.000, C 0.000 }
gfCNCPoint1[10773] = {X 182.4332, Y 57.1099, Z -1.3333, A 0.000, B 0.000, C 0.000 }
gfCNCPoint1[10774] = {X 182.5335, Y 58.0000, Z -1.3333, A 0.000, B 0.000, C 0.000 }
gfCNCPoint1[10775] = {X 182.5334, Y 58.9671, Z -1.3333, A 0.000, B 0.000, C 0.000 }
gfCNCPoint1[10776] = {X 182.4462, Y 59.7650, Z -1.3333, A 0.000, B 0.000, C 0.000 }
gfCNCPoint1[10777] = {X 182.2016, Y 60.5294, Z -1.3333, A 0.000, B 0.000, C 0.000 }
gfCNCPoint1[10778] = {X 181.8092, Y 61.2296, Z -1.3333, A 0.000, B 0.000, C 0.000 }
gfCNCPoint1[10779] = {X 209.2412, Y 91.1700, Z -1.3333, A 0.000, B 0.000, C 0.000 }
gfCNCPoint1[10780] = {X 209.9160, Y 91.8546, Z -1.3333, A 0.000, B 0.000, C 0.000 }
gfCNCPoint1[10781] = {X 210.6389, Y 92.4883, Z -1.3333, A 0.000, B 0.000, C 0.000 }
gfCNCPoint1[10782] = {X 210.9798, Y 92.7034, Z -1.3333, A 0.000, B 0.000, C 0.000 }
gfCNCPoint1[10783] = {X 211.3621, Y 92.8311, Z -1.3333, A 0.000, B 0.000, C 0.000 }
gfCNCPoint1[10784] = {X 212.3892, Y 93.0210, Z -1.3333, A 0.000, B 0.000, C 0.000 }
gfCNCPoint1[10785] = {X 213.4273, Y 93.1372, Z -1.3333, A 0.000, B 0.000, C 0.000 }
gfCNCPoint1[10786] = {X 214.4715, Y 93.0573, Z -1.3333, A 0.000, B 0.000, C 0.000 }
gfCNCPoint1[10787] = {X 215.5170, Y 92.9968, Z -1.3333, A 0.000, B 0.000, C 0.000 }
gfCNCPoint1[10788] = {X 216.2444, Y 92.9164, Z -1.3333, A 0.000, B 0.000, C 0.000 }
gfCNCPoint1[10789] = {X 216.9447, Y 92.7042, Z -1.3333, A 0.000, B 0.000, C 0.000 }
gfCNCPoint1[10790] = {X 217.5944, Y 92.3673, Z -1.3333, A 0.000, B 0.000, C 0.000 }
gfCNCPoint1[10791] = {X 223.1343, Y 88.7922, Z -1.3333, A 0.000, B 0.000, C 0.000 }
gfCNCPoint1[10792] = {X 246.5307, Y 73.8309, Z -1.3333, A 0.000, B 0.000, C 0.000 }
gfCNCPoint1[10793] = {X 221.7493, Y 64.1052, Z -1.3333, A 0.000, B 0.000, C 0.000 }
gfCNCPoint1[10794] = {X 219.9472, Y 63.5020, Z -1.3333, A 0.000, B 0.000, C 0.000 }
gfCNCPoint1[10795] = {X 218.0879, Y 63.1092, Z -1.3333, A 0.000, B 0.000, C 0.000 }
gfCNCPoint1[10796] = {X 216.1958, Y 62.9318, Z -1.3333, A 0.000, B 0.000, C 0.000 }
gfCNCPoint1[10797] = {X 215.3283, Y 62.8064, Z -1.3333, A 0.000, B 0.000, C 0.000 }
gfCNCPoint1[10798] = {X 214.5089, Y 62.4950, Z -1.3333, A 0.000, B 0.000, C 0.000 }
gfCNCPoint1[10799] = {X 213.7770, Y 62.0127, Z -1.3333, A 0.000, B 0.000, C 0.000 }
gfCNCPoint1[10800] = {X 213.1677, Y 61.3825, Z -1.3333, A 0.000, B 0.000, C 0.000 }
gfCNCPoint1[10801] = {X 212.7104, Y 60.6347, Z -1.3333, A 0.000, B 0.000, C 0.000 }
gfCNCPoint1[10802] = {X 212.4268, Y 59.8053, Z -1.3333, A 0.000, B 0.000, C 0.000 }
gfCNCPoint1[10803] = {X 212.3308, Y 58.9340, Z -1.3333, A 0.000, B 0.000, C 0.000 }
gfCNCPoint1[10804] = {X 212.3308, Y 58.0000, Z -1.3333, A 0.000, B 0.000, C 0.000 }
gfCNCPoint1[10805] = {X 212.4311, Y 57.1099, Z -1.3333, A 0.000, B 0.000, C 0.000 }
gfCNCPoint1[10806] = {X 212.7269, Y 56.2645, Z -1.3333, A 0.000, B 0.000, C 0.000 }
gfCNCPoint1[10807] = {X 213.2035, Y 55.5060, Z -1.3333, A 0.000, B 0.000, C 0.000 }
gfCNCPoint1[10808] = {X 213.8368, Y 54.8727, Z -1.3333, A 0.000, B 0.000, C 0.000 }
gfCNCPoint1[10809] = {X 214.5953, Y 54.3961, Z -1.3333, A 0.000, B 0.000, C 0.000 }
gfCNCPoint1[10810] = {X 215.4407, Y 54.1003, Z -1.3333, A 0.000, B 0.000, C 0.000 }
gfCNCPoint1[10811] = {X 216.3308, Y 54.0000, Z -1.3333, A 0.000, B 0.000, C 0.000 }
gfCNCPoint1[10812] = {X 237.2617, Y 54.0000, Z -1.3333, A 0.000, B 0.000, C 0.000 }
gfCNCPoint1[10813] = {X 238.1518, Y 54.1003, Z -1.3333, A 0.000, B 0.000, C 0.000 }
gfCNCPoint1[10814] = {X 238.9972, Y 54.3961, Z -1.3333, A 0.000, B 0.000, C 0.000 }
gfCNCPoint1[10815] = {X 239.7556, Y 54.8727, Z -1.3333, A 0.000, B 0.000, C 0.000 }
gfCNCPoint1[10816] = {X 240.3890, Y 55.5060, Z -1.3333, A 0.000, B 0.000, C 0.000 }
gfCNCPoint1[10817] = {X 240.8656, Y 56.2645, Z -1.3333, A 0.000, B 0.000, C 0.000 }
gfCNCPoint1[10818] = {X 241.1614, Y 57.1099, Z -1.3333, A 0.000, B 0.000, C 0.000 }
gfCNCPoint1[10819] = {X 241.2617, Y 58.0000, Z -1.3333, A 0.000, B 0.000, C 0.000 }
gfCNCPoint1[10820] = {X 241.2617, Y 58.4517, Z -1.3333, A 0.000, B 0.000, C 0.000 }
gfCNCPoint1[10821] = {X 247.9953, Y 61.0771, Z -1.3333, A 0.000, B 0.000, C 0.000 }
gfCNCPoint1[10822] = {X 275.9542, Y 72.1745, Z -1.3333, A 0.000, B 0.000, C 0.000 }
gfCNCPoint1[10823] = {X 275.9533, Y 63.0378, Z -1.3333, A 0.000, B 0.000, C 0.000 }
gfCNCPoint1[10824] = {X 275.9573, Y 62.9246, Z -1.3333, A 0.000, B 0.000, C 0.000 }
gfCNCPoint1[10825] = {X 275.7858, Y 62.9090, Z -1.3333, A 0.000, B 0.000, C 0.000 }
gfCNCPoint1[10826] = {X 275.6151, Y 62.8861, Z -1.3333, A 0.000, B 0.000, C 0.000 }
gfCNCPoint1[10827] = {X 274.7083, Y 62.6322, Z -1.3333, A 0.000, B 0.000, C 0.000 }
gfCNCPoint1[10828] = {X 273.8860, Y 62.1733, Z -1.3333, A 0.000, B 0.000, C 0.000 }
gfCNCPoint1[10829] = {X 273.1937, Y 61.5350, Z -1.3333, A 0.000, B 0.000, C 0.000 }
gfCNCPoint1[10830] = {X 272.6699, Y 60.7525, Z -1.3333, A 0.000, B 0.000, C 0.000 }
gfCNCPoint1[10831] = {X 272.3435, Y 59.8692, Z -1.3333, A 0.000, B 0.000, C 0.000 }
gfCNCPoint1[10832] = {X 272.2327, Y 58.9340, Z -1.3333, A 0.000, B 0.000, C 0.000 }
gfCNCPoint1[10833] = {X 272.2327, Y 58.0000, Z -1.3333, A 0.000, B 0.000, C 0.000 }
gfCNCPoint1[10834] = {X 272.3330, Y 57.1099, Z -1.3333, A 0.000, B 0.000, C 0.000 }
gfCNCPoint1[10835] = {X 272.6288, Y 56.2645, Z -1.3333, A 0.000, B 0.000, C 0.000 }
gfCNCPoint1[10836] = {X 273.1054, Y 55.5060, Z -1.3333, A 0.000, B 0.000, C 0.000 }
gfCNCPoint1[10837] = {X 273.7387, Y 54.8727, Z -1.3333, A 0.000, B 0.000, C 0.000 }
gfCNCPoint1[10838] = {X 274.4972, Y 54.3961, Z -1.3333, A 0.000, B 0.000, C 0.000 }
gfCNCPoint1[10839] = {X 275.3426, Y 54.1003, Z -1.3333, A 0.000, B 0.000, C 0.000 }
gfCNCPoint1[10840] = {X 276.2327, Y 54.0000, Z -1.3333, A 0.000, B 0.000, C 0.000 }
gfCNCPoint1[10841] = {X 292.7731, Y 54.0000, Z -1.3333, A 0.000, B 0.000, C 0.000 }
gfCNCPoint1[10842] = {X 293.6632, Y 54.1003, Z -1.3333, A 0.000, B 0.000, C 0.000 }
gfCNCPoint1[10843] = {X 294.5086, Y 54.3961, Z -1.3333, A 0.000, B 0.000, C 0.000 }
gfCNCPoint1[10844] = {X 295.2670, Y 54.8727, Z -1.3333, A 0.000, B 0.000, C 0.000 }
gfCNCPoint1[10845] = {X 295.9004, Y 55.5060, Z -1.3333, A 0.000, B 0.000, C 0.000 }
gfCNCPoint1[10846] = {X 296.3770, Y 56.2645, Z -1.3333, A 0.000, B 0.000, C 0.000 }
gfCNCPoint1[10847] = {X 296.6728, Y 57.1099, Z -1.3333, A 0.000, B 0.000, C 0.000 }
gfCNCPoint1[10848] = {X 296.7731, Y 58.0000, Z -1.3333, A 0.000, B 0.000, C 0.000 }
gfCNCPoint1[10849] = {X 296.7731, Y 58.9341, Z -1.3333, A 0.000, B 0.000, C 0.000 }
gfCNCPoint1[10850] = {X 296.6595, Y 59.8685, Z -1.3333, A 0.000, B 0.000, C 0.000 }
gfCNCPoint1[10851] = {X 296.3315, Y 60.7508, Z -1.3333, A 0.000, B 0.000, C 0.000 }
gfCNCPoint1[10852] = {X 295.8073, Y 61.5325, Z -1.3333, A 0.000, B 0.000, C 0.000 }
gfCNCPoint1[10853] = {X 295.1155, Y 62.1708, Z -1.3333, A 0.000, B 0.000, C 0.000 }
gfCNCPoint1[10854] = {X 294.2942, Y 62.6306, Z -1.3333, A 0.000, B 0.000, C 0.000 }
gfCNCPoint1[10855] = {X 293.3885, Y 62.8867, Z -1.3333, A 0.000, B 0.000, C 0.000 }
gfCNCPoint1[10856] = {X 293.2322, Y 62.9085, Z -1.3333, A 0.000, B 0.000, C 0.000 }
gfCNCPoint1[10857] = {X 293.0752, Y 62.9241, Z -1.3333, A 0.000, B 0.000, C 0.000 }
gfCNCPoint1[10858] = {X 293.0514, Y 63.1540, Z -1.3333, A 0.000, B 0.000, C 0.000 }
gfCNCPoint1[10859] = {X 293.0514, Y 92.9237, Z -1.3333, A 0.000, B 0.000, C 0.000 }
gfCNCPoint1[10860] = {X 293.0752, Y 93.0685, Z -1.3333, A 0.000, B 0.000, C 0.000 }
gfCNCPoint1[10861] = {X 293.2316, Y 93.0846, Z -1.3333, A 0.000, B 0.000, C 0.000 }
gfCNCPoint1[10862] = {X 293.3872, Y 93.1068, Z -1.3333, A 0.000, B 0.000, C 0.000 }
gfCNCPoint1[10863] = {X 294.2928, Y 93.3654, Z -1.3333, A 0.000, B 0.000, C 0.000 }
gfCNCPoint1[10864] = {X 295.1137, Y 93.8270, Z -1.3333, A 0.000, B 0.000, C 0.000 }
gfCNCPoint1[10865] = {X 295.8052, Y 94.4664, Z -1.3333, A 0.000, B 0.000, C 0.000 }
gfCNCPoint1[10866] = {X 296.3295, Y 95.2488, Z -1.3333, A 0.000, B 0.000, C 0.000 }
gfCNCPoint1[10867] = {X 296.6581, Y 96.1314, Z -1.3333, A 0.000, B 0.000, C 0.000 }
gfCNCPoint1[10868] = {X 296.7731, Y 97.0661, Z -1.3333, A 0.000, B 0.000, C 0.000 }
gfCNCPoint1[10869] = {X 296.7731, Y 98.0000, Z -1.3333, A 0.000, B 0.000, C 0.000 }
gfCNCPoint1[10870] = {X 296.6728, Y 98.8901, Z -1.3333, A 0.000, B 0.000, C 0.000 }
gfCNCPoint1[10871] = {X 296.3770, Y 99.7355, Z -1.3333, A 0.000, B 0.000, C 0.000 }
gfCNCPoint1[10872] = {X 295.9004, Y 100.4940, Z -1.3333, A 0.000, B 0.000, C 0.000 }
gfCNCPoint1[10873] = {X 295.2670, Y 101.1273, Z -1.3333, A 0.000, B 0.000, C 0.000 }
gfCNCPoint1[10874] = {X 294.5086, Y 101.6039, Z -1.3333, A 0.000, B 0.000, C 0.000 }
gfCNCPoint1[10875] = {X 293.6632, Y 101.8997, Z -1.3333, A 0.000, B 0.000, C 0.000 }
gfCNCPoint1[10876] = {X 292.7731, Y 102.0000, Z -1.3333, A 0.000, B 0.000, C 0.000 }
gfCNCPoint1[10877] = {X 276.2327, Y 102.0000, Z -1.3333, A 0.000, B 0.000, C 0.000 }
gfCNCPoint1[10878] = {X 275.3426, Y 101.8997, Z -1.3333, A 0.000, B 0.000, C 0.000 }
gfCNCPoint1[10879] = {X 274.4972, Y 101.6039, Z -1.3333, A 0.000, B 0.000, C 0.000 }
gfCNCPoint1[10880] = {X 273.7387, Y 101.1273, Z -1.3333, A 0.000, B 0.000, C 0.000 }
gfCNCPoint1[10881] = {X 273.1054, Y 100.4940, Z -1.3333, A 0.000, B 0.000, C 0.000 }
gfCNCPoint1[10882] = {X 272.6288, Y 99.7355, Z -1.3333, A 0.000, B 0.000, C 0.000 }
gfCNCPoint1[10883] = {X 272.3330, Y 98.8901, Z -1.3333, A 0.000, B 0.000, C 0.000 }
